Yaskawa INFORM job: X2_8B-21B(90,180).JBI

/JOB
//NAME X2_8B-21B(90,180)
///FOLDERNAME X2
//POS
///NPOS 939,939,939,42,0,0
///TOOL 0
///POSTYPE PULSE
///PULSE
C00000=1415,-134459,-133802,1969,12985,-79332
C00001=87080,-112473,-103627,41798,51237,-70410
C00002=91681,-107347,-99471,39221,49165,-68848
C00003=93439,-105106,-97054,38371,48113,-68361
C00004=93441,-104864,-95967,38672,47682,-68565
C00005=93504,-104969,-96260,38564,47753,-68495
C00006=95585,-102642,-95415,36914,47385,-67494
C00007=93504,-104969,-96260,38564,47753,-68495
C00008=87147,-112175,-102116,42180,50619,-70689
C00009=87145,-119394,-106475,25944,48524,-38750
C00010=91166,-110510,-101811,22693,48895,-36705
C00011=92650,-107060,-99920,21494,49065,-35962
C00012=94767,-104655,-99060,19829,49198,-34943
C00013=94484,-105085,-99259,20052,49173,-35080
C00014=93721,-102513,-96995,20598,49294,-35408
C00015=94484,-105085,-99259,20052,49173,-35080
C00016=89209,-117497,-105909,24366,48468,-37757
C00017=93166,-113214,-115710,1969,57926,-79332
C00018=93710,-106990,-108704,1652,56802,-79139
C00019=93766,-106412,-107148,1629,56140,-79127
C00020=93768,-106433,-106329,1638,55626,-79135
C00021=93918,-105383,-106173,1535,56065,-79069
C00022=94164,-101296,-104676,1361,57240,-78956
C00023=93895,-105502,-106499,1547,56205,-79076
C00024=93151,-113316,-114305,1998,57010,-79354
C00025=81072,-99391,-111155,4750,63110,-78553
C00026=81984,-95120,-104767,4287,61328,-78293
C00027=82103,-94682,-103397,4241,60705,-78273
C00028=82106,-94924,-102383,4271,59960,-78300
C00029=82089,-94934,-102578,4276,60076,-78302
C00030=82803,-90374,-100753,3806,61258,-77993
C00031=82089,-94934,-102578,4276,60076,-78302
C00032=81057,-100006,-109908,4804,62030,-78604
C00033=94004,-119945,-107122,-49530,42714,-48164
C00034=93972,-116281,-97047,-53343,39935,-45878
C00035=92833,-103149,-88492,-51302,40218,-47068
C00036=93174,-100930,-87132,-51219,40604,-47120
C00037=93174,-100493,-85792,-51770,40220,-46795
C00038=93174,-101015,-87399,-51095,40684,-47186
C00039=92955,-97894,-86230,-50180,41136,-47726
C00040=93303,-100448,-87190,-51023,40860,-47230
C00041=98055,-98607,-86499,-53149,43882,-46024
C00042=96642,-96320,-85623,-51883,43475,-46780
C00043=95342,-96864,-85830,-51299,42647,-47109
C00044=97130,-98187,-86063,-52744,43317,-46271
C00045=114545,-105110,-100746,-39625,57097,-48369
C00046=113947,-102413,-97570,-39574,56382,-48359
C00047=113947,-102278,-96691,-39772,56015,-48196
C00048=113346,-99976,-96570,-39024,56612,-48763
C00049=112899,-98120,-95866,-38597,56823,-49078
C00050=114020,-99555,-96940,-39169,57262,-48705
C00051=56302,-84822,-83054,58022,66572,-84014
C00052=58361,-85953,-83540,57558,65172,-83717
C00053=56302,-84822,-83054,58022,66572,-84014
C00054=50122,-85714,-86741,59061,71306,-84454
C00055=54195,-101901,-111197,24063,62262,-77343
C00056=67243,-111926,-101536,-21450,29925,-69540
C00057=66442,-101704,-94400,-19916,30532,-70304
C00058=66308,-99858,-92576,-19846,30336,-70336
C00059=66311,-99589,-91307,-20230,29731,-70137
C00060=66308,-99960,-93112,-19687,30597,-70418
C00061=70591,-100617,-92786,-25268,31264,-67678
C00062=70591,-100325,-91437,-25755,30647,-67424
C00063=68222,-99738,-91214,-22742,30105,-68906
C00064=70591,-100606,-92729,-25289,31242,-67667
C00065=66097,-110297,-96199,-21577,27345,-69446
C00066=65719,-107666,-92844,-21562,26575,-69447
C00067=65848,-106528,-92445,-21497,26927,-69482
C00068=65365,-110699,-93884,-21743,25627,-69354
C00069=67243,-111926,-101536,-21450,29925,-69540
C00070=68963,-41843,-96211,398,96948,48811
C00071=76932,-51697,-92360,-2602,89609,51106
C00072=71886,-45093,-85416,-705,88639,49643
C00073=71886,-45937,-84760,-705,87803,49648
C00074=71886,-44632,-85753,-705,89084,49641
C00075=68776,-90352,-95136,4313,51281,47645
C00076=68803,-86754,-93636,4241,52203,47695
C00077=68762,-92243,-95906,4353,50785,47617
C00078=77446,-64871,-91176,-8832,74282,49527
C00079=75907,-64612,-91046,-8095,74185,49034
C00080=78150,-64967,-91224,-9168,74335,49752
C00081=78150,-57569,-97635,-8943,81990,49191
C00082=68963,-41843,-96211,398,96948,48811
C00083=67385,-42511,-92598,992,94393,48367
C00084=66773,-44328,-90253,1220,92024,48175
C00085=66900,-44765,-89647,1171,91425,48205
C00086=66773,-43962,-90441,1221,92327,48178
C00087=69817,-49291,-93527,72,91467,49038
C00088=102407,-61387,-79216,-48101,75803,74984
C00089=99741,-62884,-79905,-47237,74215,74494
C00090=102407,-61387,-79216,-48101,75803,74984
C00091=71396,-101707,-96198,-105,39560,49678
C00092=71544,-99303,-95354,-247,40276,49753
C00093=71126,-105930,-97636,165,38275,49535
C00094=74447,-120283,-111838,-3099,39699,51260
C00095=57750,-84762,-113304,22338,79933,80646
C00096=38298,-117376,-123136,35520,84192,83183
C00097=31003,-114098,-105660,45955,85390,81321
C00098=32496,-116782,-107403,45795,84408,81579
C00099=34116,-118987,-108120,45640,83088,81742
C00100=33779,-118873,-108083,45678,83285,81673
C00101=33779,-118389,-106291,45736,82677,81394
C00102=33116,-116007,-107005,45711,84199,81779
C00103=35801,-87517,-89404,53765,81733,82681
C00104=39882,-82610,-88384,51436,81062,84322
C00105=41068,-84647,-89270,51225,80089,84396
C00106=40772,-84148,-89054,51277,80330,84378
C00107=40772,-84205,-87233,51414,79593,83963
C00108=38923,-82890,-88507,51652,81543,84094
C00109=36746,-57404,-73348,56767,88159,82454
C00110=45895,-41966,-67544,52307,91775,84594
C00111=46575,-44003,-68786,52133,91236,84629
C00112=46479,-43721,-68615,52158,91311,84624
C00113=46479,-44137,-67591,52124,90780,84319
C00114=45007,-43525,-68779,52515,92222,84403
C00115=28648,-44932,-73481,55068,103422,82059
C00116=23347,-70472,-95481,46672,94955,79134
C00117=23347,-70472,-95481,46672,94955,79134
C00118=34640,-80743,-102688,-17405,97112,73122
C00119=52690,-105642,-114364,-31889,95098,51390
C00120=51347,-103959,-112740,-31690,94497,51045
C00121=51347,-104280,-111882,-31650,93903,51212
C00122=54658,-102055,-112243,-32194,96275,51810
C00123=55140,-100848,-112208,-32308,96960,51798
C00124=56225,-98838,-109389,-32389,96760,52273
C00125=52710,-105778,-111943,-31798,93771,51772
C00126=54580,-102143,-110625,-32107,95358,52042
C00127=53574,-106836,-112314,-31893,93817,52092
C00128=52008,-102475,-110737,-31756,94333,51344
C00129=53574,-106836,-112314,-31893,93817,52092
C00130=61074,-96775,-114868,-33501,102293,52496
C00131=149084,-102156,-129577,-22032,95315,42360
C00132=128569,-114069,-129208,-14930,94899,36248
C00133=124702,-111484,-125119,-14131,93099,35189
C00134=123206,-111006,-122572,-13804,91571,34868
C00135=123205,-111346,-122108,-13798,91123,34918
C00136=123169,-110975,-122344,-13795,91444,34870
C00137=122647,-104244,-120003,-13724,93323,34489
C00138=123169,-110975,-122344,-13795,91444,34870
C00139=116503,-109521,-121739,-12400,90787,32743
C00140=113941,-110266,-121994,-11839,90202,31960
C00141=116503,-109521,-121739,-12400,90787,32743
C00142=121595,-114825,-128025,-13496,92670,34216
C00143=123984,-121300,-124584,-22039,85383,28695
C00144=118596,-113071,-118409,-20758,84424,26972
C00145=117828,-112575,-117002,-20585,83663,26833
C00146=117596,-112721,-116348,-20543,83158,26838
C00147=117643,-112201,-116474,-20543,83493,26797
C00148=117846,-106122,-114344,-20549,85245,26570
C00149=117643,-112201,-116474,-20543,83493,26797
C00150=125192,-113488,-115877,-22341,84450,29296
C00151=124919,-116220,-115928,-22323,83104,29449
C00152=122352,-116155,-116251,-21738,82647,28614
C00153=124919,-116220,-115928,-22323,83104,29449
C00154=123984,-121300,-124584,-22039,85383,28695
C00155=86442,-134681,-133724,19248,79211,32552
C00156=86002,-121949,-124889,19319,80358,32581
C00157=85994,-121959,-123892,19351,79775,32484
C00158=85995,-122137,-123177,19379,79272,32404
C00159=85938,-122450,-123568,19392,79360,32398
C00160=86651,-115539,-121342,19081,81262,32951
C00161=85938,-122450,-123568,19392,79360,32398
C00162=130270,-119263,-121891,-15868,79169,48216
C00163=132135,-133974,-122544,-16883,72658,49767
C00164=129371,-136174,-123179,-16117,71390,48932
C00165=132135,-133974,-122544,-16883,72658,49767
C00166=120611,-122953,-119681,-21560,80854,22535
C00167=120610,-122943,-118608,-21593,80243,22645
C00168=120610,-122853,-116921,-21650,79318,22813
C00169=120610,-122881,-117271,-21638,79506,22779
C00170=120610,-122878,-117279,-21638,79511,22778
C00171=120610,-122881,-117271,-21638,79506,22779
C00172=120610,-122873,-117198,-21640,79468,22785
C00173=120610,-122853,-117190,-21640,79473,22785
C00174=120610,-122873,-117198,-21640,79468,22785
C00175=120611,-122910,-120952,-21522,81605,22399
C00176=120612,-120891,-127143,-3106,87300,4415
C00177=120611,-122177,-124352,-3111,84925,4474
C00178=120611,-122645,-122467,-3116,83527,4507
C00179=120611,-122779,-121606,-3119,82929,4523
C00180=120611,-122697,-122159,-3117,83311,4513
C00181=120611,-122692,-122166,-3117,83318,4513
C00182=120611,-122697,-122159,-3117,83311,4513
C00183=120611,-121412,-126223,-3107,86468,4436
C00184=96873,-136971,-131305,-19961,95014,27830
C00185=53188,-122774,-119059,-34227,101931,42117
C00186=53187,-122644,-116623,-34032,100735,42492
C00187=53184,-122447,-115007,-33919,99986,42724
C00188=53180,-122268,-113886,-33849,99484,42877
C00189=53186,-122531,-115629,-33961,100272,42636
C00190=53233,-122033,-113114,-32057,113501,44659
C00191=53229,-122037,-113108,-32057,113495,44659
C00192=53233,-122033,-113114,-32057,113501,44659
C00193=53127,-122157,-112856,-34567,84618,41563
C00194=53132,-122146,-112848,-34568,84621,41564
C00195=53127,-122157,-112856,-34567,84618,41563
C00196=53124,-122720,-116247,-34514,86111,41098
C00197=68676,-133744,-131015,-10578,108811,68614
C00198=80160,-118182,-130261,41,125141,81817
C00199=80187,-122370,-123619,70,118933,81856
C00200=80183,-122639,-122398,68,118043,81854
C00201=80181,-122756,-121636,67,117515,81853
C00202=80184,-122603,-122588,68,118179,81854
C00203=80182,-122615,-122584,67,118170,81853
C00204=80184,-122603,-122588,68,118179,81854
C00205=80200,-121154,-126606,75,121396,81862
C00206=109164,-117358,-132635,7350,119146,48306
C00207=144183,-119511,-130571,15498,107286,7245
C00208=197934,-122815,-127402,28006,89082,-55776
C00209=202772,-123889,-124791,27048,85608,-54814
C00210=204705,-124106,-122314,26692,83530,-54575
C00211=204705,-124189,-120905,26732,82711,-54762
C00212=205113,-122699,-120601,26621,83104,-54520
C00213=208506,-122040,-120392,25870,82241,-53457
C00214=204510,-125657,-121990,26775,82699,-54838
C00215=204510,-125393,-124777,26704,84359,-54459
C00216=217123,-144581,-130617,26990,80795,-43719
C00217=208514,-157553,-136215,22784,79668,-13108
C00218=208514,-151468,-127497,22936,77598,-13510
C00219=209226,-147410,-126429,22728,78719,-13024
C00220=208514,-151468,-127497,22936,77598,-13510
C00221=208514,-156517,-134755,22805,79329,-13174
C00222=187736,-116553,-120968,36188,98329,-31010
C00223=144869,-104708,-130913,-697,92502,12445
C00224=97478,-100538,-119508,-25976,122096,72949
C00225=94415,-115583,-120723,-24602,114867,73486
C00226=94145,-116737,-119872,-24403,113768,73630
C00227=94090,-116915,-118863,-24267,113100,73760
C00228=94227,-118887,-121662,-24392,113788,73658
C00229=94618,-126072,-123928,-23885,111795,74261
C00230=93811,-121058,-122280,-24303,112998,73673
C00231=123165,-134656,-120887,-30393,109989,65140
C00232=122877,-135920,-118822,-30065,108215,65520
C00233=120918,-135771,-118381,-30417,107339,64954
C00234=122877,-135920,-118822,-30065,108215,65520
C00235=123434,-129548,-123417,-31323,113703,64157
C00236=126606,-101457,-128935,-16844,101795,36174
C00237=152779,-135138,-131563,-2515,76140,19155
C00238=150820,-122490,-124749,-1875,78392,18455
C00239=150097,-118368,-121531,-1645,78513,18212
C00240=150095,-118599,-120646,-1648,77850,18220
C00241=147666,-112236,-119185,-871,80184,17389
C00242=146670,-110099,-118456,-556,80825,17059
C00243=148658,-114325,-119887,-1186,79554,17722
C00244=87079,-91764,-103818,42328,107533,-9448
C00245=87027,-91004,-101788,42122,106912,-9740
C00246=89264,-90509,-101588,42089,105978,-9119
C00247=87027,-91004,-101788,42122,106912,-9740
C00248=87391,-90282,-107909,43186,109836,-8282
C00249=92115,-87061,-118989,19004,94950,3823
C00250=78975,-130870,-123203,-19746,71053,12291
C00251=74317,-97013,-111518,-17407,83606,9286
C00252=74211,-95430,-110119,-17377,83539,9259
C00253=74211,-95892,-109317,-17397,82840,9358
C00254=75305,-113551,-114600,-17838,69768,10493
C00255=78326,-111051,-111958,-19079,70114,11550
C00256=78379,-106110,-110225,-18937,71523,11339
C00257=78263,-116865,-113913,-19272,68408,11810
C00258=85880,-113569,-112821,-22054,71256,14152
C00259=85920,-114580,-110580,-22309,69503,14507
C00260=82054,-114988,-110714,-20879,68380,13249
C00261=85920,-114580,-110580,-22309,69503,14507
C00262=78975,-130870,-123203,-19746,67177,12291
C00263=159950,-115131,-126913,23322,109234,-64770
C00264=163413,-124246,-126581,22686,103792,-64589
C00265=164859,-127477,-125491,22457,101245,-64551
C00266=164857,-127553,-124648,22406,100728,-64651
C00267=164862,-127370,-126252,22506,101730,-64457
C00268=158275,-145382,-129341,21795,96649,-67831
C00269=159759,-153222,-131425,21726,93697,-67826
C00270=158275,-145382,-129341,21795,96649,-67831
C00271=157577,-144643,-126617,21696,95625,-68274
C00272=160219,-140867,-125578,21868,96138,-67212
C00273=157577,-144643,-126617,21696,95625,-68274
C00274=152631,-134238,-128202,21932,102817,-68768
C00275=146941,-123801,-133763,3444,102850,-52685
C00276=136178,-116173,-124987,-31736,84906,-22811
C00277=134413,-106132,-117362,-31242,84680,-23412
C00278=134231,-105594,-115694,-31219,83968,-23286
C00279=134230,-105863,-115134,-31239,83552,-23172
C00280=134007,-104199,-114803,-31151,84035,-23389
C00281=133473,-100630,-113499,-30965,84737,-23780
C00282=134315,-106237,-115533,-31260,83629,-23161
C00283=136272,-117460,-124003,-31807,83855,-22481
C00284=136226,-116324,-125056,-31750,84893,-22789
C00285=134474,-106353,-117504,-31259,84679,-23389
C00286=134275,-105758,-115681,-31235,83904,-23252
C00287=134274,-105987,-115198,-31252,83547,-23154
C00288=134027,-104733,-115029,-31162,83924,-23350
C00289=133465,-100971,-113658,-30966,84667,-23763
C00290=134308,-106598,-115693,-31262,83551,-23142
C00291=136269,-117902,-124178,-31812,83752,-22453
C00292=139753,-124875,-130430,-383,75663,26245
C00293=143223,-157944,-133481,5653,58679,38405
C00294=140983,-144085,-126452,6488,61628,37698
C00295=140148,-138933,-122655,6835,62006,37402
C00296=140147,-138616,-121921,6853,61719,37384
C00297=140691,-136506,-121897,6553,62737,37651
C00298=138669,-131542,-120459,7325,64564,37004
C00299=140691,-136506,-121897,6553,62737,37651
C00300=145148,-139028,-124584,4588,62787,39337
C00301=159973,-92454,-110285,-14523,90938,48717
C00302=158765,-97223,-112137,-14224,89465,48492
C00303=159973,-92454,-110285,-14523,90938,48717
C00304=164681,-91509,-114703,-15696,94847,49769
C00305=142525,-105883,-132766,7713,103357,60336
C00306=90751,-115691,-121566,36045,104861,61043
C00307=92920,-122587,-117773,35137,99152,60047
C00308=93124,-123070,-117553,35091,98753,60003
C00309=93124,-123008,-116878,35050,98435,59900
C00310=93160,-123063,-117190,35068,98555,59953
C00311=95752,-125144,-117838,34977,96947,60505
C00312=93160,-123063,-117190,35068,98555,59953
C00313=92038,-109836,-114685,38536,89453,57060
C00314=86810,-100893,-104585,47463,92019,56975
C00315=88449,-102594,-103600,47188,90148,56855
C00316=88449,-102618,-102426,47172,89639,56610
C00317=88449,-102603,-103366,47184,90046,56806
C00318=85133,-99388,-102162,47637,92393,56350
C00319=85168,-99488,-101153,47595,91912,56132
C00320=86978,-101259,-101820,47360,90627,56378
C00321=84037,-98201,-102123,47804,93363,56297
C00322=108771,-112096,-123986,16313,85813,59347
C00323=109769,-112695,-132242,3132,99947,61138
C00324=127404,-127157,-120795,-27540,73197,60883
C00325=120526,-123085,-115007,-25540,69700,59025
C00326=119461,-122312,-114032,-25210,69192,58723
C00327=119461,-122116,-113003,-25293,68708,58832
C00328=119461,-122312,-114032,-25210,69192,58723
C00329=94655,-112249,-115827,1041,75214,51009
C00330=93364,-111129,-115444,1499,75574,50577
C00331=121213,-123445,-114215,-25873,69302,59387
C00332=127714,-127278,-119628,-27738,72603,61150
C00333=140848,-129628,-128054,-17424,84805,27418
C00334=127903,-106251,-120637,-17388,91568,15860
C00335=124887,-98361,-114445,-16717,91208,14907
C00336=124614,-94849,-112077,-16660,91489,14780
C00337=117832,-103976,-115449,-15062,87719,13014
C00338=118209,-109888,-118953,-15141,86934,13233
C00339=120968,-118649,-124805,-15800,86569,14208
C00340=112726,-101228,-128594,-1890,90279,-15897
C00341=102865,-105549,-130121,1361,88970,-18873
C00342=85416,-143080,-122146,23399,58401,-32529
C00343=89847,-131888,-116792,20882,59491,-30436
C00344=92362,-125061,-113696,19444,60385,-29236
C00345=93061,-123120,-113350,17672,61903,-28193
C00346=94553,-118505,-112300,14045,65420,-26024
C00347=98668,-108930,-110937,8182,72602,-22159
C00348=97558,-114678,-114533,8498,72116,-22521
C00349=94805,-124749,-120489,9597,70928,-23580
C00350=89899,-115674,-129227,15589,81503,-27304
C00351=94000,-113154,-130859,-1035,116659,75004
C00352=93721,-118000,-129934,-5060,122177,74127
C00353=93715,-120352,-127357,-4900,119392,74256
C00354=95323,-119775,-124837,-4467,118233,74917
C00355=88228,-120746,-125279,-6046,117555,72254
C00356=93725,-120284,-127319,-4898,119404,74259
C00357=93731,-117931,-129895,-5059,122189,74130
C00358=92605,-107385,-114202,42080,118626,78084
C00359=94957,-117308,-114744,40643,113912,77125
C00360=98035,-118959,-113942,40650,111458,77555
C00361=97377,-118969,-113658,40508,111623,77311
C00362=92838,-119913,-111612,39284,112339,75456
C00363=89330,-129662,-113469,38848,107684,75257
C00364=90618,-118755,-112828,39302,114392,75239
C00365=88476,-109244,-112462,40625,118981,76164
C00366=73726,-95231,-122050,23824,117115,78775
C00367=68964,-113071,-130294,-19412,109419,80322
C00368=55630,-112625,-122011,-35520,97927,81697
C00369=52390,-118820,-120628,-34805,93310,81881
C00370=47903,-104132,-115503,-31781,99116,78849
C00371=50154,-103283,-114443,-33074,100204,79243
C00372=58838,-110339,-112590,-36869,98506,82639
C00373=58731,-119232,-119174,-35403,94943,83913
C00374=59872,-116629,-120975,-35716,97415,83571
C00375=61517,-148095,-119735,-48293,75564,80066
C00376=56687,-146008,-116451,-48020,72337,79248
C00377=54787,-145656,-114853,-48003,70776,79074
C00378=55742,-144545,-112808,-48270,70818,79550
C00379=55476,-147094,-115701,-48129,70996,79318
C00380=61520,-147186,-118480,-48348,75358,80173
C00381=69196,-132761,-125763,-48066,87564,77891
C00382=67178,-112107,-133350,9560,121946,71499
C00383=53652,-115588,-130730,10921,119132,80041
C00384=53631,-118653,-128170,10572,116038,79726
C00385=49979,-127897,-130457,9357,109364,77840
C00386=56749,-116857,-125794,10963,115112,80794
C00387=55258,-116620,-125691,10759,115364,80266
C00388=57875,-118021,-126871,3069,115075,80163
C00389=60441,-120565,-127584,-682,114000,80575
C00390=56047,-119336,-124870,-1283,112953,79038
C00391=53493,-120154,-126714,-1639,113579,78070
C00392=53512,-117734,-129516,-1682,116546,78033
C00393=64263,-112177,-127274,-18013,116425,52133
C00394=53349,-113292,-116223,-34708,105130,41711
C00395=53347,-113647,-113946,-34435,103813,42137
C00396=52619,-113100,-112715,-34376,103127,42055
C00397=57761,-122997,-112011,-36249,97635,45734
C00398=53343,-113729,-112902,-34324,103242,42318
C00399=53345,-113489,-115217,-34581,104530,41905
C00400=83368,-135406,-127982,-43757,111124,-24122
C00401=107112,-148704,-121184,-48737,110155,-73723
C00402=107085,-142005,-111593,-48000,108472,-72828
C00403=107084,-140010,-108705,-47787,107957,-72557
C00404=87341,-136498,-115496,-38254,104619,-81025
C00405=107242,-151301,-127119,1131,113743,-57617
C00406=97067,-157300,-128671,2718,111508,-55981
C00407=110320,-141463,-116471,39094,91497,-45920
C00408=107133,-145289,-116877,40503,90261,-47122
C00409=107139,-146938,-119316,40521,90762,-46927
C00410=81304,-146505,-131302,46256,99624,-33732
C00411=42290,-135810,-134986,6789,56953,43412
C00412=53482,-111499,-99357,5283,31563,44884
C00413=53488,-110753,-96932,5448,30458,44798
C00414=53767,-110832,-96596,5125,30193,44961
C00415=53784,-109802,-93724,5302,28956,44868
C00416=54077,-108600,-90505,5126,27581,44957
C00417=54077,-108600,-90505,5126,27581,44957
C00418=53472,-108968,-91791,5862,28222,44586
C00419=53466,-109889,-94290,5675,29282,44681
C00420=93748,-113667,-111432,-27227,62688,41579
C00421=93751,-113561,-109328,-27520,61581,41869
C00422=94298,-111463,-107612,-27765,61782,42046
C00423=94581,-111188,-102370,-28702,59144,42896
C00424=93743,-112935,-104615,-28181,59286,42489
C00425=93741,-113330,-106821,-27872,60309,42206
C00426=53707,-103235,-126817,3349,90409,72793
C00427=53694,-107630,-124107,3352,86490,72685
C00428=54249,-109117,-122940,3188,84989,72821
C00429=53889,-108493,-122718,3296,85190,72712
C00430=53934,-108401,-122669,3281,85203,72729
C00431=53898,-108487,-122690,3292,85171,72715
C00432=53735,-107561,-124050,3339,86489,72698
C00433=53748,-103173,-126762,3336,90406,72805
C00434=24309,-104032,-127063,11845,92683,63842
C00435=14692,-96968,-103634,28347,84848,56264
C00436=69737,67118,16632,42575,112328,80617
C00437=69765,65699,24866,49286,110081,81190
C00438=67763,57248,15205,49930,112177,81338
C00439=66597,45471,2237,49732,108456,84264
C00440=65732,29116,-14706,47956,102511,88210
C00441=64654,15507,-27591,48359,103674,88304
C00442=64160,11579,-31342,48521,104111,88301
C00443=61960,-11325,-50587,48960,105231,87855
C00444=62752,-490,-42039,50927,111117,85502
C00445=59065,9442,-33802,52095,101706,84381
C00446=72891,31150,-30442,36756,97726,81673
C00447=90877,-16324,-74885,22437,92008,81813
C00448=102330,-22799,-82036,-11222,88832,73278
C00449=48313,-118911,-129560,-19207,92704,27073
C00450=53495,-110604,-121584,-20154,93282,28749
C00451=52758,-114738,-121214,-19966,90894,28894
C00452=53577,-108529,-119024,-20154,92819,28853
C00453=53441,-111570,-120070,-20107,91929,28955
C00454=54259,-112639,-122766,-20278,93161,29031
C00455=53522,-108468,-123882,-20258,95652,28360
C00456=66910,-101677,-117691,-1645,82254,-17515
C00457=66905,-103395,-115374,-1652,79946,-17486
C00458=66781,-102668,-113970,-1597,79454,-17514
C00459=66805,-103111,-114336,-1620,79451,-17514
C00460=68500,-103754,-114391,-2206,79196,-16952
C00461=69944,-105966,-109421,-11944,70678,-17306
C00462=66783,-105788,-110032,-11324,70201,-18483
C00463=66785,-105108,-112553,-11207,72068,-18659
C00464=34610,-119076,-126707,31995,89279,-47352
C00465=26693,-119602,-105841,51320,82883,-62074
C00466=26676,-118953,-103885,51392,82336,-62389
C00467=27513,-117883,-103390,51295,82023,-62119
C00468=27155,-116250,-99936,51446,81403,-62657
C00469=26666,-118021,-101324,51491,81640,-62785
C00470=26683,-118745,-103309,51412,82173,-62476
C00471=26741,-121947,-116429,51038,86269,-60171
C00472=80158,-111738,-121779,46707,81282,33331
C00473=80124,-114295,-114082,47454,77096,31277
C00474=80115,-114367,-110881,47781,75720,30584
C00475=82694,-112805,-110607,45433,76546,32096
C00476=79416,-116776,-110373,48221,75031,29878
C00477=80052,-114603,-110983,47806,75713,30548
C00478=80061,-114542,-114188,47480,77086,31241
C00479=80063,-113108,-120040,30435,104055,77976
C00480=80050,-114212,-116860,30086,101864,77373
C00481=79953,-112412,-114936,30056,101673,77283
C00482=79896,-114545,-111990,35011,85373,77209
C00483=80002,-114499,-112021,34994,85367,77250
C00484=80418,-112503,-109508,36583,80313,77299
C00485=80029,-114714,-111597,36713,80437,77233
C00486=82440,-93132,-104306,35744,84828,79668
C00487=83142,-90791,-100833,35602,83775,79606
C00488=86899,-75258,-94009,34443,85431,81601
C00489=81341,-82881,-101909,35963,88366,80388
C00490=80042,-114535,-115070,36542,82240,77847
C00491=80040,-111621,-122742,8414,85267,41918
C00492=80035,-113457,-119567,8450,82400,41723
C00493=81653,-127299,-120603,7413,72175,41563
C00494=80787,-111090,-118654,-2680,86591,53574
C00495=79816,-113282,-119312,-2452,85841,53272
C00496=79371,-114754,-119577,-3684,84607,55046
C00497=80002,-113603,-119620,-10752,83390,63441
C00498=80006,-103113,-128729,-10775,94202,62513
C00499=39776,-103787,-110683,21075,62663,-59255
C00500=39766,-104399,-107995,21452,60825,-59622
C00501=42409,-98411,-106612,17292,64181,-58311
C00502=40224,-103973,-106702,21316,60174,-59568
C00503=40236,-103975,-106617,21326,60117,-59576
C00504=39744,-104425,-108009,21464,60826,-59630
C00505=39754,-103814,-110697,21087,62664,-59263
C00506=47977,-106691,-119962,23629,83327,-62671
C00507=66867,-99660,-121232,22132,99220,-62132
C00508=66851,-102572,-118810,21937,96446,-62653
C00509=75734,-133384,-127933,14237,79030,-52956
C00510=72894,-135572,-127272,15029,78051,-54067
C00511=68354,-138260,-126704,16229,77252,-55778
C00512=51043,-132166,-118737,30188,81179,-60892
C00513=66851,-103895,-117201,21852,94891,-62938
C00514=66868,-101493,-119792,22004,97521,-62449
C00515=74321,-107832,-126985,-11736,80239,-61811
C00516=66584,-114412,-108983,-34198,49386,-64476
C00517=66581,-113854,-105403,-35147,47795,-63826
C00518=60037,-123864,-103215,-32979,33373,-60846
C00519=66685,-112635,-100589,-36483,45924,-62949
C00520=66087,-122535,-98001,-45910,35159,-56780
C00521=66087,-122589,-97589,-46197,34963,-56624
C00522=66567,-113311,-102857,-35821,46729,-63375
C00523=66569,-114089,-106515,-34851,48256,-64025
C00524=66614,-114312,-115902,-32344,53032,-65825
C00525=26293,-124733,-123676,-35115,86081,-77095
C00526=26278,-124914,-120130,-35186,84196,-76502
C00527=26896,-123210,-118103,-35309,84144,-76233
C00528=26306,-121290,-117658,-35177,84490,-76583
C00529=26301,-124893,-120124,-35190,84211,-76498
C00530=26317,-124710,-123669,-35119,86096,-77090
C00531=26368,-124828,-121889,-39154,95960,-78120
C00532=26350,-124746,-118556,-38992,94373,-77544
C00533=26743,-123924,-117047,-38976,94149,-77295
C00534=25994,-118731,-112182,-38918,93559,-77400
C00535=26347,-124286,-115407,-38884,93032,-77056
C00536=26365,-124761,-118865,-39006,94524,-77592
C00537=26264,-124528,-116402,-47920,86072,-68134
C00538=26249,-123768,-112787,-47988,84810,-67516
C00539=26243,-123374,-111311,-48022,84325,-67278
C00540=27566,-121809,-108978,-48187,84599,-66758
C00541=26232,-123227,-110778,-48035,84146,-67194
C00542=26247,-124165,-114452,-47952,85370,-67795
C00543=82585,-123093,-118421,-52491,64599,-59558
C00544=107155,-118824,-102398,-58122,50036,-52281
C00545=107155,-117467,-98958,-59145,49269,-51564
C00546=97405,-116506,-103900,-42249,48003,-50997
C00547=106070,-119659,-109558,-10435,43390,-62985
C00548=106582,-120227,-109824,-10893,43331,-62728
C00549=108221,-120478,-109947,-12283,43512,-61940
C00550=107366,-119665,-105766,-8068,39033,-71395
C00551=107169,-120346,-107141,-7797,39493,-71540
C00552=108433,-119625,-117514,-7930,46308,-71537
C00553=107111,-122100,-111275,-39348,45202,-56077
C00554=107109,-117760,-98763,-43179,41028,-53713
C00555=107588,-117193,-97805,-43718,41045,-53392
C00556=106524,-118597,-102582,-12234,37369,-61918
C00557=94589,-117778,-102277,12815,37699,-75547
C00558=102638,-119985,-97555,45693,41122,-79392
C00559=107127,-114270,-91297,56630,43098,-80056
C00560=101354,-119078,-102486,55464,49091,-79315
C00561=93612,-109275,-133010,-12113,75674,-64968
C00562=74458,-81913,-116300,-25886,107898,-47202
C00563=74285,-84923,-113224,-25351,104735,-46539
C00564=81136,-80920,-107787,-32217,106507,-45804
C00565=73205,-70766,-105026,-26930,108371,-55320
C00566=67013,-54988,-96314,-28913,109390,-56440
C00567=64326,-60619,-98517,-27945,103439,-54917
C00568=60588,-58283,-100875,-23679,106756,-51616
C00569=60637,-54628,-103477,-24231,109960,-52288
C00570=76657,-70403,-83915,-51355,64349,-40407
C00571=74830,-68241,-74355,-53953,55282,-38932
C00572=73110,-62379,-68708,-53436,54020,-39148
C00573=73205,-61459,-68120,-53411,54142,-39173
C00574=37101,-67408,-75626,25719,44355,-77225
C00575=80454,-89253,-85222,-18196,36589,-55164
C00576=82537,-90732,-84998,-19061,34673,-56543
C00577=81508,-95500,-88175,-18158,33969,-56993
C00578=81043,-103588,-94156,-17854,33413,-57140
C00579=82846,-88179,-88219,-41798,48730,-43563
C00580=81818,-81213,-82326,-41198,48211,-43888
C00581=79628,-80184,-80995,-37948,46295,-45131
C00582=64054,-84747,-85294,-4301,39779,-58682
C00583=75679,-87820,-86686,-15780,40506,-52732
C00584=49490,-70910,-80897,34287,57978,-66074
C00585=46339,-68382,-80235,37741,61555,-66618
C00586=42699,-70655,-83815,39176,63943,-67342
C00587=43803,-67144,-92021,36183,69839,-64523
C00588=86906,-70734,-117845,-25978,101850,-24881
C00589=194376,-118372,-116958,-36622,58194,75254
C00590=187943,-106127,-101715,-33777,52366,74665
C00591=187951,-105693,-98645,-34509,50978,75202
C00592=188084,-106418,-97655,-35041,50218,75578
C00593=188317,-106012,-97596,-35084,50459,75600
C00594=188444,-106426,-98768,-20061,46138,60546
C00595=187923,-105820,-99644,-19403,46817,60144
C00596=187914,-106157,-102495,-18928,48312,59826
C00597=188021,-109107,-91072,-54887,40419,77132
C00598=188025,-108188,-88773,-55807,39869,77674
C00599=188027,-107805,-87846,-56180,39654,77892
C00600=188036,-107761,-87717,-56242,39627,77928
C00601=188035,-108145,-88644,-55869,39841,77710
C00602=188030,-109068,-90945,-54948,40390,77168
C00603=188015,-114130,-110744,-41340,72657,75143
C00604=188018,-113864,-107763,-41683,71368,75679
C00605=188019,-113684,-106544,-41824,70871,75888
C00606=188009,-113674,-106577,-41816,70886,75877
C00607=188008,-113852,-107795,-41674,71383,75668
C00608=188005,-114114,-110775,-41332,72673,75132
C00609=187933,-113872,-110928,-18210,58720,57176
C00610=187882,-113256,-105308,719,43762,42538
C00611=187896,-112711,-102669,725,42418,42533
C00612=188420,-113689,-102063,268,41535,42791
C00613=188115,-112866,-98519,1306,37390,42477
C00614=187899,-111729,-99017,1491,38283,42378
C00615=187886,-112431,-101600,1465,39511,42393
C00616=192869,-127835,-120494,-22551,66263,53872
C00617=188079,-122619,-114609,-40714,83609,61664
C00618=188077,-122103,-112045,-40794,82601,62056
C00619=187715,-122511,-111198,-41935,87054,59703
C00620=187919,-121855,-110458,-41952,87063,59791
C00621=187909,-121652,-109146,-41964,86526,60005
C00622=188106,-121566,-109755,-41972,86936,59927
C00623=188110,-122188,-112187,-41960,87826,59570
C00624=188058,-121965,-125191,-40549,88870,59628
C00625=104402,-90439,-123637,-22599,88102,-26907
C00626=80407,-121901,-119741,-18448,66455,-46046
C00627=80400,-121844,-116068,-18757,64334,-45697
C00628=80537,-121388,-114459,-18932,63649,-45528
C00629=79603,-120238,-114067,-18464,63768,-45911
C00630=80475,-121542,-115946,-18779,64427,-45684
C00631=80482,-121578,-119613,-18469,66554,-46034
C00632=85156,-144709,-129107,21632,59402,-64028
C00633=93856,-120445,-109825,39450,57641,-70752
C00634=92040,-118150,-105716,42198,57852,-71483
C00635=84290,-104454,-97866,49611,66426,-72991
C00636=89339,-123311,-104077,50362,59795,-74015
C00637=89538,-124434,-104337,50489,59412,-74133
C00638=89538,-124434,-104337,50489,59412,-74133
C00639=93820,-118277,-102341,40471,46353,-72255
C00640=93828,-119232,-105178,39715,47322,-71755
C00641=93822,-120125,-107980,28359,52237,-38282
C00642=93816,-119582,-106091,28689,51458,-38525
C00643=93586,-119120,-105470,28875,51409,-38650
C00644=93805,-118409,-102529,29499,49391,-39302
C00645=93820,-119862,-107056,29266,59584,-40856
C00646=93823,-120114,-107958,29147,59957,-40747
C00647=93830,-120670,-110185,28854,60909,-40473
C00648=63807,-119595,-131717,32346,77391,-31957
C00649=66677,-122882,-119460,9954,65715,31882
C00650=66675,-122709,-116301,10101,63887,31721
C00651=67233,-123478,-115304,9930,62823,31836
C00652=66931,-123352,-121183,-9496,81515,37764
C00653=66923,-123307,-121544,-9492,81753,37743
C00654=68643,-124975,-117174,-29306,103015,42901
C00655=66675,-122499,-114776,-33395,107690,42822
C00656=66677,-122795,-117228,-33681,108831,42458
C00657=66720,-122114,-124411,-34847,112827,41144
C00658=15972,-110889,-128286,10965,59905,43045
C00659=15972,-110889,-128286,10965,59905,43045
C00660=101389,-60822,-75148,-6919,68546,70102
C00661=115790,69230,64798,8053,66131,71909
C00662=120688,105020,73307,12402,84846,73777
C00663=120868,103639,75593,12409,82749,73629
C00664=115729,87511,60668,24910,80664,72140
C00665=115729,87728,62416,24969,79785,71953
C00666=115729,87559,61087,24923,80450,72095
C00667=115791,92601,67435,24996,79233,71857
C00668=115791,92884,68992,25055,78493,71699
C00669=115775,91432,67152,25030,78849,71769
C00670=115791,92590,67368,24993,79266,71865
C00671=126095,92435,63058,5152,80409,74477
C00672=126453,92655,64525,5082,79598,74565
C00673=125768,92396,64197,5232,79709,74335
C00674=126453,92544,63242,5072,80328,74595
C00675=120228,112105,88453,12614,79365,73063
C00676=120053,112844,85327,12571,81642,73235
C00677=120830,71540,61874,4756,55589,66514
C00678=120535,76858,72419,5134,51864,66212
C00679=120418,79487,77321,5314,50212,66075
C00680=120418,81305,81326,5435,48689,65991
C00681=120418,79487,77321,5314,50212,66075
C00682=121101,73566,71896,4942,50464,66384
C00683=120640,77942,77238,5256,49458,66131
C00684=121101,73566,71896,4942,50464,66384
C00685=121222,71175,67349,4775,52021,66512
C00686=121527,63287,45853,4167,61152,67017
C00687=121222,53388,35819,-506,60999,72680
C00688=120886,47658,32975,-2750,58873,75677
C00689=120357,43570,36815,-5865,53609,79607
C00690=120357,44263,39245,-5952,52477,79673
C00691=120357,43570,36815,-5865,53609,79607
C00692=121171,39511,33217,-6288,53799,79936
C00693=121171,39929,34748,-6347,53075,79981
C00694=120657,42834,37803,-6102,52651,79790
C00695=121171,39929,34748,-6347,53075,79981
C00696=121307,38577,31710,-6326,54255,79965
C00697=121648,35573,24568,-6294,57116,79932
C00698=109578,65571,33028,8923,84264,70984
C00699=101389,-60822,-75148,-6919,68546,70102
C00700=96929,-90691,-89138,-5080,61517,23019
C00701=109818,-91701,-74936,-12505,53754,-21374
C00702=124678,-6429,-38037,-6148,92089,-49038
C00703=133997,38575,-5386,-4879,105902,-64390
C00704=134430,35731,-4221,-4855,103756,-64161
C00705=134605,34666,-3678,-4847,102887,-64068
C00706=134604,34193,-2477,-4825,101908,-64030
C00707=134605,34666,-3678,-4847,102887,-64068
C00708=133324,38381,1851,-4717,101326,-64430
C00709=133984,36157,-436,-4773,101627,-64224
C00710=133324,38381,1851,-4717,101326,-64430
C00711=132740,42105,45,-4739,104308,-64739
C00712=149381,11612,-10676,-29411,77480,-58612
C00713=147438,22168,3080,-29176,74144,-58502
C00714=146667,27061,10007,-29185,72341,-58335
C00715=146666,27163,11157,-29282,71765,-58183
C00716=146667,27014,9351,-29131,72675,-58422
C00717=147917,24004,8167,-29618,72393,-57848
C00718=149025,12105,-2903,-29837,73391,-57674
C00719=148491,19843,4212,-29741,72852,-57742
C00720=149112,19141,-2052,-29482,76126,-58364
C00721=148788,18564,-14441,-28797,82460,-60100
C00722=147017,27605,-1759,-28452,79091,-59917
C00723=146805,27803,661,-28506,77793,-59674
C00724=146803,27699,1600,-28565,77235,-59535
C00725=146805,27874,109,-28472,78126,-59757
C00726=148390,24338,-1607,-29025,77984,-59121
C00727=147556,26192,183,-28786,77573,-59333
C00728=148390,24338,-1607,-29025,77984,-59121
C00729=149162,23542,-7999,-28991,81344,-59682
C00730=129846,-17397,-52274,-16165,101048,-68229
C00731=103949,-6271,-30701,-7884,96105,-76175
C00732=94102,16895,-5866,-4380,94047,-79161
C00733=94024,14878,-3719,-4358,91692,-79105
C00734=93993,14152,-2780,-4351,90742,-79083
C00735=93993,14253,-1030,-4349,89719,-79047
C00736=93993,14152,-2780,-4351,90742,-79083
C00737=93685,20015,4382,-4321,89334,-79138
C00738=93881,17120,1686,-4338,89515,-79078
C00739=93685,20015,4382,-4321,89334,-79138
C00740=93796,22544,1176,-4343,92603,-79213
C00741=95224,-25687,-42365,-27028,60157,-72238
C00742=94111,-23276,-36997,-26973,57954,-72128
C00743=93676,-22245,-34794,-26967,57075,-72081
C00744=93677,-22196,-33100,-27266,56165,-71832
C00745=93676,-22245,-34794,-26967,57075,-72081
C00746=94165,-26445,-35973,-27662,55954,-71554
C00747=93910,-23559,-33944,-27450,56079,-71704
C00748=94165,-26445,-35973,-27662,55954,-71554
C00749=95768,-30118,-43626,-27714,58991,-71694
C00750=97625,-41604,-59467,-17173,89706,8843
C00751=96114,-37688,-53918,-16886,88057,8555
C00752=95526,-36022,-51615,-16777,87400,8443
C00753=95527,-36150,-50037,-16784,86406,8579
C00754=95526,-36022,-51615,-16777,87400,8443
C00755=95532,-36183,-50637,-16782,86745,8534
C00756=95234,-33170,-48668,-16723,87008,8396
C00757=95532,-36183,-50637,-16782,86745,8534
C00758=95504,-36095,-50208,-16778,86530,8554
C00759=93996,-36675,-50581,-16493,86163,8084
C00760=95504,-36095,-50208,-16778,86530,8554
C00761=97625,-41604,-59467,-17173,89706,8843
C00762=101873,-77751,-87156,-42969,63075,-62474
C00763=95937,-74809,-81328,-40948,58735,-63434
C00764=95565,-74583,-80935,-40815,58468,-63500
C00765=95566,-74620,-79294,-41227,57681,-63141
C00766=95565,-74583,-80935,-40815,58468,-63500
C00767=98755,-73227,-80296,-42221,60183,-62682
C00768=98803,-73638,-78797,-42678,59356,-62269
C00769=96868,-74481,-79195,-41849,58298,-62761
C00770=98803,-73638,-78797,-42678,59356,-62269
C00771=97163,-69666,-76891,-41573,59236,-63045
C00772=96752,-66139,-75134,-41097,59602,-63417
C00773=97163,-69666,-76891,-41573,59236,-63045
C00774=101873,-77751,-87156,-42969,63075,-62474
C00775=126113,-49786,-51573,-51544,90004,-55144
C00776=123973,-50127,-48217,-51392,87374,-54806
C00777=123267,-50126,-46982,-51347,86566,-54726
C00778=118449,-34614,-37258,-50921,85079,-56444
C00779=119272,-35479,-39244,-50973,86038,-56539
C00780=121232,-35158,-42579,-51146,88553,-56901
C00781=111145,-57425,-62081,-41633,61582,-55088
C00782=109620,-53993,-56645,-41578,59663,-54986
C00783=109182,-52175,-54253,-41602,59047,-54926
C00784=105694,-54761,-55728,-40263,57099,-55829
C00785=106107,-56401,-57979,-40230,57706,-55889
C00786=107578,-60042,-63488,-40293,59558,-55964
C00787=93331,-25535,-46307,-22677,87971,-72102
C00788=84242,-5399,-27465,-11713,100257,-81196
C00789=83743,-8192,-25851,-11599,97806,-81134
C00790=83568,-8790,-24556,-11558,96698,-81088
C00791=80825,-8752,-24536,-11465,96320,-81994
C00792=80973,-8366,-25985,-11504,97411,-82047
C00793=81511,-5615,-27635,-11617,99868,-82095
C00794=103949,-6271,-30701,-7884,96105,-76175
C00795=129846,-17397,-52274,-16165,101048,-68229
C00796=163642,29140,5761,-44799,70700,-52559
C00797=162591,31494,11671,-45064,68427,-51999
C00798=162048,30394,11874,-43983,65447,-51631
C00799=161982,31813,14334,-41708,59650,-50819
C00800=161467,24519,6374,-40573,59309,-51272
C00801=161788,23282,1722,-39913,61178,-51925
C00802=148843,20256,-8268,-42580,75292,-58905
C00803=147687,21461,-3477,-42608,73008,-58456
C00804=147474,22713,-827,-42735,72168,-58194
C00805=145829,17703,-5538,-42117,71635,-58722
C00806=146103,16605,-8013,-42018,72487,-58958
C00807=147273,15378,-12798,-41999,74773,-59389
C00808=132879,31978,-11069,-11402,105457,-66436
C00809=133021,29093,-9797,-11280,103253,-66180
C00810=131898,46229,9833,-9962,110180,-66921
C00811=130688,40255,3261,-9867,109174,-67217
C00812=130053,42231,5661,-10091,111027,-67639
C00813=131193,25278,-13529,-11136,103347,-66799
C00814=131063,28208,-14820,-11259,105588,-67051
C00815=112468,-32306,-55652,-4896,84919,-46156
C00816=96808,-82585,-76071,-53,68600,-46133
C00817=69953,-63335,-76496,8026,68297,-36882
C00818=96929,-90691,-89138,-5080,61517,23019
C00819=101389,-60822,-75148,-6919,68546,70102
C00820=109578,66950,51259,9202,73878,70224
C00821=119285,73548,61078,7759,54489,67872
C00822=119140,78931,71700,8230,50768,67516
C00823=119625,58082,57992,11126,34581,65932
C00824=123364,68268,69491,7525,32771,67988
C00825=122687,69615,57970,5984,54089,69256
C00826=122770,54503,36545,5592,59480,69583
C00827=119074,82203,59752,14757,75142,72556
C00828=112473,77653,55392,16315,76732,70397
C00829=112597,64720,47818,22234,69078,68724
C00830=113195,66142,49473,22093,68650,68874
C00831=113258,68857,52652,22154,68111,68793
C00832=116388,75351,60395,21391,65952,69596
C00833=116375,72151,56555,21287,66626,69721
C00834=116824,73080,57665,21174,66318,69837
C00835=121396,72779,51526,8459,68942,71502
C00836=127130,57447,36738,757,68697,35525
C00837=129893,63235,47621,-3557,65457,33128
C00838=128808,60089,44122,-3143,65953,32716
C00839=130205,57581,36634,-4742,69462,32000
C00840=130312,54578,33992,-4779,69550,32035
C00841=129992,46081,35923,-20239,67004,-8502
C00842=121835,41418,34711,-6021,59386,-22657
C00843=117745,46484,42710,5309,56994,-25598
C00844=117421,45985,43643,5502,56187,-25765
C00845=128073,50557,47782,-20949,62737,-7811
C00846=128141,51586,49590,-20554,61962,-8032
C00847=121273,40131,39499,-4242,51746,-24031
C00848=122651,35401,27095,-8965,61652,-19959
C00849=109578,66950,51259,9202,73878,70224
C00850=101389,-60822,-75148,-6919,68546,70102
C00851=96929,-90691,-89138,-5080,61517,23019
C00852=93242,-104717,-83164,-3670,50463,-28203
C00853=113023,-47673,-50887,-12494,73990,-34579
C00854=92156,-22649,-39625,-10516,94476,-60392
C00855=92549,-23820,-36378,-10508,91967,-60047
C00856=93168,-23682,-34836,-10551,91183,-59771
C00857=95681,-22921,-34071,-10762,91434,-58934
C00858=94898,-22950,-35761,-10710,92338,-59280
C00859=94492,-21797,-39017,-10723,94837,-59633
C00860=92575,-26977,-42679,-21088,73618,-56030
C00861=92430,-25186,-37423,-21282,71416,-55682
C00862=92878,-24238,-35435,-21526,70842,-55408
C00863=96065,-22906,-34163,-23638,71815,-54341
C00864=95477,-23933,-36320,-23344,72386,-54682
C00865=95719,-25683,-41558,-23174,74597,-55037
C00866=111616,-56743,-62949,-22039,72011,-39056
C00867=96929,-90691,-89138,-5080,61517,-27168
C00868=96929,-90691,-89138,-5080,61517,23019
C00869=101389,-60822,-75148,-6919,68546,70102
C00870=109578,66950,51259,9202,73878,70224
C00871=108278,48890,46404,6655,48460,73563
C00872=108252,54023,56228,7048,45078,73302
C00873=108060,40798,52110,13776,28764,70729
C00874=112800,50045,60477,7453,29903,74191
C00875=112495,52250,52136,4220,46380,75358
C00876=112766,56024,54314,4011,46966,75508
C00877=103660,28975,43016,-10311,30529,75473
C00878=104692,35200,60863,-30413,16065,83251
C00879=105089,39423,66918,-34170,14880,85035
C00880=103103,37348,64656,-29541,14457,82654
C00881=100412,37194,55383,-7603,26828,73795
C00882=100998,29868,43914,-7479,30147,73786
C00883=109578,66950,51259,9202,73878,70224
C00884=101389,-60822,-75148,-6919,68546,70102
C00885=96929,-90691,-89138,-5080,61517,23019
C00886=92414,-106749,-81881,-3283,48598,-28500
C00887=109112,-55837,-56038,-6601,71444,-37060
C00888=90570,-23240,-39845,1682,91658,-61068
C00889=90349,-1837,-19216,4288,101242,-62233
C00890=89876,4658,-11592,5336,104467,-62228
C00891=91883,5295,-10855,6364,104142,-61464
C00892=95291,-22836,-35623,1093,89189,-59526
C00893=94239,-22001,-38963,1226,91687,-59852
C00894=90424,-29050,-43505,-3763,58999,-61302
C00895=86008,-21130,-36360,6353,62529,-61992
C00896=86680,-19135,-33236,6051,61587,-61792
C00897=89871,-18454,-32736,4367,61424,-60601
C00898=95351,-24457,-36663,-6763,57473,-59317
C00899=94707,-27619,-42528,-6252,59394,-59681
C00900=109011,-26713,-50438,-8452,98222,-74634
C00901=131236,23776,-19025,3434,93964,-64709
C00902=130664,38162,-3482,6829,99038,-64158
C00903=130670,46363,8576,7678,101442,-63891
C00904=134671,48665,11259,6610,97243,-62896
C00905=136543,32349,-6519,2125,90508,-63120
C00906=135803,33584,-9338,2313,92894,-63310
C00907=159001,-16036,-30877,-42377,70566,-51510
C00908=152463,-28313,-30724,-35893,55196,-47069
C00909=153151,-16160,-21724,-35569,61642,-49446
C00910=157385,-8578,-13959,-39473,60379,-46999
C00911=158653,-15121,-22520,-39743,62752,-48156
C00912=161766,-5301,-16021,-44095,69224,-49591
C00913=91964,-16840,-43330,-6553,97397,-80206
C00914=99312,-50897,-61026,-22837,72179,-74454
C00915=98138,-49989,-56545,-22703,69739,-74412
C00916=107037,-51945,-50657,-37198,66142,-70452
C00917=99628,-21060,-40506,-23543,91538,-75534
C00918=101911,-27523,-44444,-25592,91744,-74763
C00919=98969,-20169,-40937,-21673,97560,-76394
C00920=97496,-21660,-46096,-18879,96544,-76387
C00921=97638,-23312,-49453,-18962,97729,-76524
C00922=81141,-50558,-66105,-12803,46081,-75388
C00923=80687,-46119,-60183,-12697,44679,-75401
C00924=80513,-44339,-57785,-12667,44105,-75401
C00925=80516,-44488,-54802,-13120,42239,-75121
C00926=80690,-46329,-57233,-13145,42803,-75122
C00927=81145,-50923,-63237,-13239,44177,-75109
C00928=83601,15534,-39616,-9664,96262,-77072
C00929=80484,90945,50155,-4324,118905,-78550
C00930=80490,84570,45509,-4303,118490,-78531
C00931=80493,82108,43801,-4293,118276,-78521
C00932=80495,81630,46278,-4216,116511,-78452
C00933=80492,84058,47940,-4226,116735,-78462
C00934=83493,53381,-2692,-9637,111099,-78940
C00935=91945,-14209,-43630,-9790,83010,-75128
C00936=107113,-96096,-84434,-15453,68738,-68360
C00937=10907,-117335,-90652,18762,63715,59495
C00938=15972,-110889,-128286,10965,59905,43045
BC00000=48813,501269,1075139
BC00001=366895,287876,1075139
BC00002=366895,287876,1075139
BC00003=366895,287876,1075139
BC00004=366895,287876,1075139
BC00005=366895,287876,1075139
BC00006=366895,287876,1075139
BC00007=366895,287876,1075139
BC00008=366895,287876,1075139
BC00009=333040,294697,1075139
BC00010=333040,294697,1075139
BC00011=333040,294697,1075139
BC00012=333040,294697,1075139
BC00013=333040,294697,1075139
BC00014=333040,294697,1075139
BC00015=333040,294697,1075139
BC00016=333040,294697,1075139
BC00017=358075,287887,1075139
BC00018=358075,287887,1075139
BC00019=358075,287887,1075139
BC00020=358075,287887,1075139
BC00021=358075,287887,1075139
BC00022=358075,287887,1075139
BC00023=358075,287887,1075139
BC00024=358075,287887,1075139
BC00025=398158,296006,1075139
BC00026=398158,296006,1075139
BC00027=398158,296006,1075139
BC00028=398158,296006,1075139
BC00029=398158,296006,1075139
BC00030=398158,296006,1075139
BC00031=398158,296006,1075139
BC00032=398158,296006,1075139
BC00033=264887,408839,1075139
BC00034=264887,408839,1075139
BC00035=264888,408840,1075136
BC00036=264888,408840,1075135
BC00037=264888,408840,1075135
BC00038=264888,408840,1075132
BC00039=264888,408840,1075132
BC00040=264888,408840,1075132
BC00041=264888,408840,1075132
BC00042=264888,408840,1075132
BC00043=264888,408840,1075128
BC00044=264887,408839,1075139
BC00045=301248,414295,1075139
BC00046=301248,414295,1075139
BC00047=301248,414295,1075139
BC00048=301248,414295,1075139
BC00049=301248,414295,1075139
BC00050=301248,414295,1075139
BC00051=301248,414295,1075139
BC00052=301248,414295,1075139
BC00053=301248,414295,1075139
BC00054=301248,414295,1075139
BC00055=274219,403900,1075139
BC00056=238656,390224,1075139
BC00057=238656,390224,1075139
BC00058=238656,390224,1075139
BC00059=238656,390224,1075139
BC00060=238656,390224,1075139
BC00061=238656,390224,1075139
BC00062=238656,390224,1075139
BC00063=238656,390224,1075139
BC00064=238656,390225,1075135
BC00065=238656,390225,1075135
BC00066=238656,390224,1075139
BC00067=238656,390224,1075139
BC00068=238656,390224,1075139
BC00069=238656,390224,1075139
BC00070=318247,439655,1075139
BC00071=318247,439655,1075139
BC00072=318247,439655,1075139
BC00073=318247,439655,1075139
BC00074=318247,439655,1075139
BC00075=318247,439655,1075139
BC00076=318247,439655,1075139
BC00077=318247,439655,1075139
BC00078=318247,439655,1075139
BC00079=318247,439655,1075139
BC00080=318247,439655,1075139
BC00081=318247,439655,1075139
BC00082=318247,439655,1075139
BC00083=318247,439655,1075139
BC00084=318247,439655,1075139
BC00085=318247,439655,1075139
BC00086=318247,439655,1075139
BC00087=318247,439655,1075139
BC00088=318247,439655,1075139
BC00089=318247,439655,1075139
BC00090=318247,439655,1075139
BC00091=318247,439655,1075139
BC00092=318247,439655,1075139
BC00093=318247,439655,1075139
BC00094=318247,439655,1075139
BC00095=377098,439655,1075139
BC00096=397798,439655,1075139
BC00097=397798,439655,1075139
BC00098=397798,439655,1075139
BC00099=397798,439655,1075139
BC00100=397798,439655,1075139
BC00101=397798,439655,1075139
BC00102=397798,439655,1075139
BC00103=397798,439655,1075139
BC00104=397798,439655,1075139
BC00105=397798,439655,1075139
BC00106=397798,439655,1075139
BC00107=397798,439655,1075139
BC00108=397798,439655,1075139
BC00109=397798,439655,1075139
BC00110=397798,439655,1075139
BC00111=397798,439655,1075139
BC00112=397798,439655,1075139
BC00113=397798,439655,1075139
BC00114=397798,439655,1075139
BC00115=397798,439655,1075139
BC00116=390344,433324,1075139
BC00117=390344,433324,1075139
BC00118=323680,511522,1075139
BC00119=296258,353406,1075139
BC00120=296258,353406,1075139
BC00121=296258,353406,1075139
BC00122=296258,353406,1075139
BC00123=296258,353406,1075139
BC00124=296258,353406,1075139
BC00125=296258,353406,1075139
BC00126=296258,353406,1075139
BC00127=296258,353406,1075139
BC00128=296258,353406,1075139
BC00129=296258,353406,1075139
BC00130=296258,353406,1075139
BC00131=312199,290121,1075139
BC00132=312199,245824,1075139
BC00133=312199,245824,1075139
BC00134=312199,245824,1075139
BC00135=312199,245824,1075139
BC00136=312199,245824,1075139
BC00137=312199,245824,1075139
BC00138=312199,245824,1075139
BC00139=312199,245824,1075139
BC00140=312199,245824,1075139
BC00141=312199,245824,1075139
BC00142=312199,245824,1075139
BC00143=259283,251148,1075139
BC00144=259283,251148,1075139
BC00145=259283,251148,1075139
BC00146=259283,251148,1075139
BC00147=259283,251148,1075139
BC00148=259283,251148,1075139
BC00149=259283,251148,1075139
BC00150=259283,251148,1075139
BC00151=259283,251148,1075139
BC00152=259283,251148,1075139
BC00153=259283,251148,1075139
BC00154=259283,251148,1075139
BC00155=211515,238198,1075139
BC00156=211515,238198,1075139
BC00157=211515,238198,1075139
BC00158=211515,238198,1075139
BC00159=211515,238198,1075139
BC00160=211515,238198,1075139
BC00161=211515,238198,1075139
BC00162=211515,238198,1075139
BC00163=211515,238198,1075139
BC00164=211515,238198,1075139
BC00165=211515,238198,1075139
BC00166=182487,238237,1075139
BC00167=184353,236726,1075139
BC00168=184353,236710,1075139
BC00169=184317,236583,1075139
BC00170=184881,233559,1075139
BC00171=184317,236583,1075139
BC00172=184735,236445,1075139
BC00173=187871,236988,1075139
BC00174=184735,236445,1075139
BC00175=178206,241731,1075139
BC00176=185188,240150,1075139
BC00177=186084,235310,1075139
BC00178=186442,233366,1075138
BC00179=186443,233357,1075139
BC00180=186562,233334,1075139
BC00181=187125,230310,1075139
BC00182=186562,233334,1075139
BC00183=185308,240110,1075139
BC00184=153065,191986,1075139
BC00185=123072,128894,1075139
BC00186=126316,134328,1075139
BC00187=127614,136496,1075139
BC00188=127614,136486,1075139
BC00189=127614,136502,1075139
BC00190=153737,125360,1075139
BC00191=152136,128016,1075139
BC00192=153737,125360,1075139
BC00193=104350,151955,1075139
BC00194=107104,153499,1075139
BC00195=104350,151955,1075139
BC00196=97474,145929,1075139
BC00197=140327,144391,1075139
BC00198=158627,143734,1075139
BC00199=155448,149073,1075139
BC00200=155090,149654,1075139
BC00201=155090,149646,1075139
BC00202=155272,149742,1075139
BC00203=153671,152398,1075139
BC00204=155272,149742,1075139
BC00205=158875,143812,1075139
BC00206=211321,196495,1075139
BC00207=274607,206177,1075139
BC00208=371745,147058,1075139
BC00209=371745,147058,1075139
BC00210=371745,147058,1075139
BC00211=371745,147058,1075139
BC00212=371745,147058,1075139
BC00213=371745,147058,1075139
BC00214=371745,147058,1075139
BC00215=371745,147058,1075139
BC00216=371745,147058,1075139
BC00217=371745,147058,1075139
BC00218=371745,147058,1075139
BC00219=371745,147058,1075139
BC00220=371745,147058,1075139
BC00221=371745,147058,1075139
BC00222=371745,147058,1075139
BC00223=314169,251254,1075139
BC00224=247655,219498,1075139
BC00225=247655,219498,1075139
BC00226=247655,219498,1075139
BC00227=247655,219498,1075139
BC00228=247655,219498,1075139
BC00229=247655,219498,1075139
BC00230=247655,219498,1075139
BC00231=247655,219498,1075139
BC00232=247655,219498,1075139
BC00233=247655,219498,1075139
BC00234=247655,219498,1075139
BC00235=247655,219498,1075139
BC00236=303021,318054,1075139
BC00237=380976,369454,1075139
BC00238=380976,369454,1075139
BC00239=380976,369454,1075139
BC00240=380976,369454,1075139
BC00241=380976,369454,1075139
BC00242=380976,369454,1075139
BC00243=380976,369454,1075139
BC00244=380976,369454,1075139
BC00245=380976,369454,1075139
BC00246=380976,369454,1075139
BC00247=380976,369454,1075139
BC00248=380976,369454,1075139
BC00249=275240,377785,1075139
BC00250=125700,292206,1075139
BC00251=125700,292206,1075139
BC00252=125700,292206,1075139
BC00253=125700,292206,1075139
BC00254=125700,292206,1075139
BC00255=125700,292206,1075138
BC00256=125700,292206,1075135
BC00257=125700,292206,1075139
BC00258=125700,292206,1075139
BC00259=125700,292206,1075139
BC00260=125700,292206,1075139
BC00261=125700,292206,1075139
BC00262=125700,292206,1075139
BC00263=325003,367566,1075193
BC00264=325003,367566,1075193
BC00265=325003,367566,1075193
BC00266=325003,367566,1075193
BC00267=325003,367566,1075193
BC00268=325003,367566,1075193
BC00269=325003,367566,1075193
BC00270=325003,367566,1075193
BC00271=325003,367566,1075193
BC00272=325003,367566,1075193
BC00273=325003,367566,1075193
BC00274=325003,367566,1075193
BC00275=240651,318179,1075174
BC00276=81319,224890,1075139
BC00277=81319,224890,1075139
BC00278=81319,224890,1075139
BC00279=81319,224890,1075139
BC00280=81319,224890,1075139
BC00281=81319,224890,1075139
BC00282=81319,224890,1075139
BC00283=81319,224890,1075139
BC00284=39875,217643,1075139
BC00285=39875,217643,1075139
BC00286=39875,217643,1075139
BC00287=39875,217643,1075139
BC00288=39875,217643,1075139
BC00289=39875,217643,1075139
BC00290=39875,217643,1075139
BC00291=39875,217643,1075139
BC00292=126048,247985,1075139
BC00293=145702,238926,1075139
BC00294=145702,238926,1075139
BC00295=145702,238926,1075139
BC00296=145702,238926,1075139
BC00297=145702,238926,1075139
BC00298=145702,238926,1075139
BC00299=145702,238926,1075139
BC00300=145702,238926,1075139
BC00301=145702,238926,1075139
BC00302=145702,238926,1075139
BC00303=145702,238926,1075139
BC00304=145702,238926,1075139
BC00305=127177,276102,1075139
BC00306=75481,322634,1075139
BC00307=75481,322634,1075139
BC00308=75481,322634,1075139
BC00309=75481,322634,1075139
BC00310=75481,322634,1075139
BC00311=75481,322634,1075139
BC00312=75481,322634,1075139
BC00313=75481,322634,1075139
BC00314=75481,322634,1075139
BC00315=75481,322634,1075139
BC00316=75481,322634,1075139
BC00317=75481,322634,1075139
BC00318=75481,322634,1075139
BC00319=75481,322634,1075139
BC00320=75481,322634,1075139
BC00321=75481,322634,1075139
BC00322=75481,322634,1075139
BC00323=58814,337696,1075139
BC00324=43258,351755,1075139
BC00325=43258,351755,1075139
BC00326=43258,351755,1075139
BC00327=43258,351755,1075139
BC00328=43258,351755,1075139
BC00329=43258,351755,1075139
BC00330=43258,351755,1075139
BC00331=43258,351755,1075139
BC00332=43258,351755,1075139
BC00333=191423,293819,1075139
BC00334=209577,315616,1075139
BC00335=209577,315616,1075139
BC00336=209577,315616,1075139
BC00337=209577,315616,1075135
BC00338=209577,315616,1075139
BC00339=209577,315616,1075139
BC00340=209200,339183,1075139
BC00341=226850,335636,1075139
BC00342=228819,334245,1075139
BC00343=228819,334245,1075139
BC00344=228818,334247,1075135
BC00345=228818,334246,1075136
BC00346=228819,334245,1075139
BC00347=228819,334245,1075139
BC00348=228819,334245,1075139
BC00349=228819,334245,1075139
BC00350=228819,334245,1075139
BC00351=212667,203752,1075139
BC00352=212667,185592,1075139
BC00353=212231,190237,1075139
BC00354=212130,191331,1075135
BC00355=214778,193391,1075138
BC00356=222170,195981,1075139
BC00357=222606,191336,1075139
BC00358=293461,217046,1075139
BC00359=293461,217046,1075139
BC00360=293461,217046,1075139
BC00361=293461,217046,1075139
BC00362=293461,217046,1075139
BC00363=293461,217046,1075139
BC00364=293461,217046,1075139
BC00365=293461,217046,1075139
BC00366=248761,215697,1075139
BC00367=147608,172175,1075139
BC00368=124934,156734,1075139
BC00369=124934,156734,1075139
BC00370=124934,156734,1075139
BC00371=124934,156734,1075139
BC00372=124934,156734,1075139
BC00373=124934,156734,1075139
BC00374=124934,156734,1075139
BC00375=106662,143944,1075139
BC00376=106662,143944,1075139
BC00377=106662,143944,1075139
BC00378=106662,143944,1075139
BC00379=106662,143944,1075139
BC00380=106662,143944,1075139
BC00381=106662,155705,1075139
BC00382=288347,238792,1075139
BC00383=319864,257821,1075139
BC00384=316187,259932,1075139
BC00385=314717,260776,1075138
BC00386=314716,260777,1075139
BC00387=294125,249227,1075139
BC00388=285335,240623,1075139
BC00389=280828,236212,1075139
BC00390=254340,221178,1075136
BC00391=253980,219316,1075139
BC00392=256761,216362,1075139
BC00393=224898,195450,1075139
BC00394=193391,175353,1075139
BC00395=196536,180842,1075139
BC00396=197049,181737,1075139
BC00397=197381,182312,1075139
BC00398=196536,180831,1075139
BC00399=193391,175343,1075139
BC00400=170860,158975,1075139
BC00401=152991,145993,1075139
BC00402=152991,145993,1075139
BC00403=155583,151896,1075139
BC00404=156620,154258,1075139
BC00405=230582,164381,1075139
BC00406=176880,134401,1075139
BC00407=222677,176979,1075139
BC00408=228168,179508,1075139
BC00409=235185,179594,1075139
BC00410=242581,209775,1075139
BC00411=282664,373339,1075139
BC00412=287377,415944,1075139
BC00413=293850,413917,1075139
BC00414=296439,413107,1075139
BC00415=296321,413021,1075139
BC00416=296321,413021,1075139
BC00417=296321,413021,1075139
BC00418=293584,413723,1075139
BC00419=287111,415750,1075139
BC00420=265157,384983,1075139
BC00421=271825,383261,1075139
BC00422=274492,382572,1075139
BC00423=274492,382572,1075139
BC00424=271826,383216,1075139
BC00425=265158,384938,1075139
BC00426=347759,380452,1075139
BC00427=348420,380650,1075139
BC00428=348684,380729,1075139
BC00429=352817,383042,1075139
BC00430=364797,389762,1075139
BC00431=368926,392082,1075139
BC00432=368661,392003,1075139
BC00433=368000,391805,1075139
BC00434=368000,391805,1075139
BC00435=374651,423539,1075139
BC00436=391328,503109,1075139
BC00437=391328,503109,1075139
BC00438=391328,503109,1075139
BC00439=391328,503109,1075139
BC00440=391328,503109,1075139
BC00441=391328,503109,1075139
BC00442=391328,503109,1075139
BC00443=391328,503109,1075139
BC00444=391328,503108,1075138
BC00445=391328,503109,1075139
BC00446=391328,503109,1075139
BC00447=391328,503109,1075139
BC00448=358857,503109,1075139
BC00449=250155,294085,1075139
BC00450=255354,296197,1075139
BC00451=257433,297042,1075139
BC00452=259835,293058,1075139
BC00453=270486,275398,1075139
BC00454=268406,274554,1075139
BC00455=263207,272441,1075139
BC00456=251679,365603,1075139
BC00457=253900,360561,1075139
BC00458=254788,358544,1075138
BC00459=231432,345511,1075139
BC00460=231432,345511,1075139
BC00461=193281,329322,1075139
BC00462=188554,329982,1075139
BC00463=185285,334773,1075139
BC00464=261316,356567,1075139
BC00465=297096,366823,1075139
BC00466=293507,360766,1075139
BC00467=292071,358344,1075139
BC00468=292072,358325,1075139
BC00469=293507,360744,1075139
BC00470=297096,366801,1075139
BC00471=297096,366823,1075139
BC00472=112329,235363,1075139
BC00473=112329,235363,1075139
BC00474=111530,230597,1075139
BC00475=111210,228691,1075139
BC00476=63682,220459,1075139
BC00477=64002,222365,1075139
BC00478=64801,227131,1075139
BC00479=55513,330800,1075139
BC00480=51579,332061,1075139
BC00481=50005,332565,1075139
BC00482=45879,356917,1075139
BC00483=46055,340308,1075139
BC00484=43971,345622,1075139
BC00485=45459,346376,1075139
BC00486=45459,346376,1075139
BC00487=45459,346376,1075139
BC00488=45459,346376,1075139
BC00489=45459,346376,1075139
BC00490=49366,347783,1075139
BC00491=32175,334569,1075139
BC00492=35183,333207,1075139
BC00493=36386,332662,1075139
BC00494=24154,317654,1075139
BC00495=24100,334244,1075139
BC00496=21697,333868,1075139
BC00497=10090,331721,1075139
BC00498=7091,330415,1075139
BC00499=124149,231378,1075139
BC00500=124461,225905,1075139
BC00501=124586,223716,1075139
BC00502=119883,222901,1075139
BC00503=114643,221993,1075139
BC00504=114518,224182,1075139
BC00505=114206,229656,1075139
BC00506=169481,226749,1075139
BC00507=218439,224175,1075139
BC00508=214415,222148,1075139
BC00509=212806,221337,1075139
BC00510=212806,221337,1075139
BC00511=212806,221337,1075139
BC00512=212806,221337,1075139
BC00513=218328,226790,1075139
BC00514=222352,228818,1075139
BC00515=147308,231841,1075139
BC00516=86334,206095,1075139
BC00517=90701,204719,1075139
BC00518=92225,204354,1075139
BC00519=87933,207931,1075139
BC00520=87933,207931,1075139
BC00521=87933,207931,1075139
BC00522=86186,208482,1075139
BC00523=81819,209859,1075139
BC00524=86334,206095,1075139
BC00525=118170,307260,1075139
BC00526=118297,311064,1075139
BC00527=118347,312586,1075139
BC00528=127335,312613,1075139
BC00529=127284,311091,1075139
BC00530=127157,307287,1075139
BC00531=149515,294377,1075139
BC00532=148233,298842,1075139
BC00533=148018,300627,1075139
BC00534=150070,300618,1075139
BC00535=152272,298825,1075139
BC00536=153553,294359,1075139
BC00537=119286,287990,1075139
BC00538=119424,292460,1075139
BC00539=119479,294248,1075139
BC00540=115958,294219,1075139
BC00541=115903,292431,1075139
BC00542=115765,287961,1075139
BC00543=206834,274416,1075139
BC00544=246621,268498,1075139
BC00545=251225,265487,1075139
BC00546=253066,264282,1075139
BC00547=305610,287542,1075139
BC00548=289507,284753,1075139
BC00549=289507,284753,1075139
BC00550=265981,288415,1075136
BC00551=265766,290089,1075139
BC00552=265230,294276,1075139
BC00553=152789,271435,1075139
BC00554=155628,267409,1075139
BC00555=156764,265799,1075139
BC00556=187125,277004,1075139
BC00557=135483,267954,1075139
BC00558=183860,266265,1075139
BC00559=204587,267200,1075139
BC00560=210051,271155,1075139
BC00561=285477,353851,1075139
BC00562=322658,411530,1075139
BC00563=322658,411530,1075139
BC00564=322658,411530,1075139
BC00565=322658,411530,1075139
BC00566=322658,411530,1075139
BC00567=322658,411530,1075139
BC00568=322658,411530,1075139
BC00569=322658,411530,1075139
BC00570=272539,420945,1075139
BC00571=266463,422086,1075139
BC00572=266463,422086,1075139
BC00573=267463,419870,1071329
BC00574=266783,420774,1075139
BC00575=266463,422086,1075139
BC00576=266463,422086,1075139
BC00577=266463,422086,1075139
BC00578=266463,422086,1075139
BC00579=235968,403705,1075139
BC00580=235968,403705,1075139
BC00581=235968,403705,1075139
BC00582=235968,403705,1075139
BC00583=235968,403705,1075139
BC00584=235968,403705,1075139
BC00585=235968,403705,1075139
BC00586=235968,403705,1075139
BC00587=237187,402741,1075139
BC00588=295006,362715,1075139
BC00589=205685,258924,1075139
BC00590=204796,257891,1075139
BC00591=205655,252480,1075139
BC00592=205999,250316,1075139
BC00593=202530,248347,1075139
BC00594=218277,237314,1075139
BC00595=218450,239623,1075139
BC00596=218882,245393,1075139
BC00597=188210,264707,1075139
BC00598=189282,258005,1075139
BC00599=189712,255325,1075139
BC00600=185359,252882,1075139
BC00601=184930,255563,1075139
BC00602=183858,262264,1075139
BC00603=163240,249581,1075139
BC00604=166744,245232,1075139
BC00605=168145,243492,1075139
BC00606=172944,246185,1075139
BC00607=171543,247924,1075139
BC00608=168039,252273,1075139
BC00609=205588,237933,1075139
BC00610=237359,225800,1075139
BC00611=234842,220095,1075139
BC00612=233835,217813,1075139
BC00613=237392,219487,1075139
BC00614=238410,221660,1075139
BC00615=241123,227449,1075139
BC00616=186179,231259,1075139
BC00617=137514,234633,1075139
BC00618=142324,230418,1075139
BC00619=135201,224052,1075139
BC00620=135201,224052,1075139
BC00621=134384,223577,1075139
BC00622=132247,225161,1075139
BC00623=126952,229147,1075139
BC00624=137514,234633,1075139
BC00625=284854,339782,1075139
BC00626=323088,248514,1075139
BC00627=324420,245120,1075139
BC00628=324953,243763,1075139
BC00629=379843,253270,1075139
BC00630=379310,254627,1075139
BC00631=377978,258021,1075139
BC00632=387009,264306,1075139
BC00633=391855,267678,1075139
BC00634=387117,263921,1075139
BC00635=386182,263175,1075138
BC00636=386182,263175,1075138
BC00637=386182,263175,1075138
BC00638=386182,263175,1075138
BC00639=364780,283240,1075139
BC00640=368854,287926,1075139
BC00641=358141,287701,1075139
BC00642=354860,281457,1075139
BC00643=353548,278959,1075139
BC00644=349122,282807,1075139
BC00645=357556,273175,1075139
BC00646=359162,275355,1075139
BC00647=363177,280805,1075139
BC00648=322742,336521,1075139
BC00649=135423,234905,1075139
BC00650=139936,232261,1075139
BC00651=141741,231203,1075139
BC00652=133024,192287,1075139
BC00653=133049,212626,1075139
BC00654=142080,160489,1075139
BC00655=142682,147059,1075139
BC00656=139311,141641,1075139
BC00657=142682,147059,1075139
BC00658=21198,517278,1075139
BC00659=21198,517278,429866
BC00660=66799,465991,419725
BC00661=110224,417152,337633
BC00662=124980,400556,122247
BC00663=124980,400556,122247
BC00664=124980,400556,122247
BC00665=124980,400556,122247
BC00666=124980,400556,122247
BC00667=124980,400556,122247
BC00668=124980,400556,122247
BC00669=124980,400556,122247
BC00670=124980,400556,122247
BC00671=124980,400556,122247
BC00672=124980,400556,122247
BC00673=124980,400556,122247
BC00674=124980,400556,122247
BC00675=124980,400556,122247
BC00676=124980,400556,122247
BC00677=136713,400556,283945
BC00678=136713,400556,283945
BC00679=136713,400556,283945
BC00680=136713,400556,283945
BC00681=136713,400556,283945
BC00682=136713,400556,283945
BC00683=136713,400556,283945
BC00684=136713,400556,283945
BC00685=136713,400556,283945
BC00686=136713,400556,232066
BC00687=148065,400556,238331
BC00688=154841,400556,249660
BC00689=163178,400556,279134
BC00690=163178,400556,279134
BC00691=163178,400556,279134
BC00692=163178,400556,279134
BC00693=163178,400556,279134
BC00694=163178,400556,279134
BC00695=163178,400556,279134
BC00696=163178,400556,279134
BC00697=163178,400556,279134
BC00698=110224,417152,230098
BC00699=66799,465991,419725
BC00700=66799,519251,419725
BC00701=252749,519251,277295
BC00702=296498,463393,186341
BC00703=322792,429821,131675
BC00704=322792,429821,131675
BC00705=322792,429821,131675
BC00706=322792,429821,131675
BC00707=322792,429821,131675
BC00708=322792,429821,131675
BC00709=322792,429821,131675
BC00710=322792,429821,131675
BC00711=322792,429821,131675
BC00712=303662,400556,204886
BC00713=303662,411227,204886
BC00714=303662,415917,204886
BC00715=303662,415917,204886
BC00716=303662,415917,204886
BC00717=303662,415917,204886
BC00718=303662,400556,204886
BC00719=303662,411314,204886
BC00720=303662,412604,204886
BC00721=343990,442081,139026
BC00722=343990,437458,139026
BC00723=343990,437458,139026
BC00724=343990,437458,139026
BC00725=343990,437458,139026
BC00726=343990,437458,139026
BC00727=343990,437458,139026
BC00728=343990,437458,139026
BC00729=343990,437458,139026
BC00730=300917,439314,218872
BC00731=283877,440048,250459
BC00732=276304,440374,264498
BC00733=276304,440374,264498
BC00734=276304,440374,264498
BC00735=276304,440374,264498
BC00736=276304,440374,264498
BC00737=276304,440374,264498
BC00738=276304,440374,264498
BC00739=276304,440374,264498
BC00740=276304,440374,264498
BC00741=248841,426339,138655
BC00742=248841,426339,138655
BC00743=248841,426339,138655
BC00744=248841,426339,138655
BC00745=248841,426339,138655
BC00746=248841,426339,138655
BC00747=248841,426339,138655
BC00748=248841,426339,138655
BC00749=248841,426339,138655
BC00750=287848,400556,132674
BC00751=287848,400556,132674
BC00752=287848,400556,132674
BC00753=287848,400556,132674
BC00754=287848,400556,132674
BC00755=287848,400556,132674
BC00756=287848,400556,132674
BC00757=287848,400556,132674
BC00758=287848,400556,132674
BC00759=287848,400556,132674
BC00760=287848,400556,132674
BC00761=287848,400556,132674
BC00762=279813,400556,17
BC00763=279813,400556,17
BC00764=279813,400556,17
BC00765=279813,400556,17
BC00766=279813,400556,17
BC00767=279813,400556,17
BC00768=279813,400556,17
BC00769=279813,400556,17
BC00770=279813,400556,17
BC00771=279813,400556,17
BC00772=279813,400556,17
BC00773=279813,400556,17
BC00774=279813,400556,17
BC00775=312308,400556,158769
BC00776=312308,400556,158769
BC00777=312308,400556,158768
BC00778=312308,400556,158769
BC00779=312308,400556,158769
BC00780=312308,400556,158769
BC00781=303066,421715,105063
BC00782=303066,421715,105063
BC00783=303066,421715,105063
BC00784=303066,421715,105063
BC00785=303066,421715,105063
BC00786=303066,421715,105063
BC00787=287852,408667,183289
BC00788=278394,400556,231917
BC00789=278394,400556,231917
BC00790=278394,400556,231917
BC00791=278394,400556,231917
BC00792=278394,400556,231917
BC00793=278394,400556,231917
BC00794=283877,440048,250459
BC00795=300917,439314,218872
BC00796=328923,417583,120701
BC00797=328923,417583,120701
BC00798=328923,417583,120701
BC00799=328923,417583,120701
BC00800=328923,417583,120701
BC00801=328923,417583,120701
BC00802=337213,453034,95368
BC00803=337213,453034,95368
BC00804=337213,453034,95368
BC00805=337213,453034,95368
BC00806=337213,453034,95368
BC00807=337213,453034,95368
BC00808=318162,429946,122343
BC00809=318162,429946,122343
BC00810=318162,429946,122343
BC00811=318162,429946,122343
BC00812=318162,429946,122343
BC00813=318162,429946,122343
BC00814=318162,429946,122343
BC00815=257174,478061,205827
BC00816=245597,487118,221641
BC00817=204965,519251,277295
BC00818=66799,519251,419725
BC00819=66799,465991,419725
BC00820=110224,417152,337633
BC00821=118787,400556,240422
BC00822=118787,400556,240422
BC00823=118787,400556,240422
BC00824=118787,400556,240422
BC00825=118787,400556,240422
BC00826=118787,400556,240422
BC00827=130243,400556,198340
BC00828=110693,400556,198340
BC00829=113235,400556,198340
BC00830=113235,400556,198340
BC00831=113235,400556,198340
BC00832=113235,400556,198340
BC00833=113235,400556,198340
BC00834=113235,400556,198340
BC00835=113235,400556,198340
BC00836=113235,400556,198340
BC00837=113235,400556,198340
BC00838=113235,400556,198340
BC00839=113235,400556,198340
BC00840=113235,400556,228006
BC00841=113235,400556,280256
BC00842=113235,400556,280254
BC00843=113235,400556,280254
BC00844=113235,400556,280254
BC00845=113235,400556,280254
BC00846=113235,400556,280254
BC00847=113235,400556,280254
BC00848=113235,400556,280254
BC00849=110224,417152,337633
BC00850=66799,465991,419725
BC00851=66799,519251,419725
BC00852=252749,519251,277295
BC00853=271419,473397,262334
BC00854=298317,407335,240779
BC00855=298317,407335,240779
BC00856=298317,407335,240779
BC00857=298317,407335,240779
BC00858=298317,407335,240779
BC00859=298317,407335,240779
BC00860=277580,417028,190893
BC00861=277580,417028,190893
BC00862=277580,417028,190893
BC00863=277580,417028,190893
BC00864=277580,417028,190893
BC00865=277580,417028,190893
BC00866=268077,456148,223959
BC00867=252749,519251,277295
BC00868=66799,519251,419725
BC00869=66799,465991,419725
BC00870=110224,417152,337633
BC00871=116529,400556,319233
BC00872=116529,400556,319233
BC00873=116529,400556,319233
BC00874=116529,400556,319233
BC00875=116529,400556,319233
BC00876=116529,400556,319233
BC00877=104242,400556,379272
BC00878=104242,400556,379272
BC00879=104242,400556,379272
BC00880=104242,400556,379272
BC00881=104242,400556,379272
BC00882=104242,400556,379272
BC00883=110224,417152,337633
BC00884=66799,465991,419725
BC00885=66799,539969,419725
BC00886=252749,519251,277295
BC00887=268071,466646,260861
BC00888=286658,402854,240926
BC00889=286659,402854,240926
BC00890=286659,402854,240926
BC00891=286659,402854,240926
BC00892=286658,402854,240926
BC00893=286658,402854,240926
BC00894=267093,432072,158905
BC00895=267093,432072,158905
BC00896=267093,432072,158905
BC00897=267093,432072,158905
BC00898=267093,432072,158905
BC00899=267093,432072,158905
BC00900=283877,440048,250459
BC00901=320500,429384,110898
BC00902=320500,429384,110898
BC00903=320500,429384,110898
BC00904=320500,429384,110898
BC00905=320500,429384,110898
BC00906=320500,429384,110898
BC00907=331313,400556,191260
BC00908=331313,400556,191260
BC00909=331313,400556,191260
BC00910=331313,400556,191260
BC00911=331313,400556,191260
BC00912=331313,400556,191260
BC00913=244057,440048,250459
BC00914=292954,400556,136487
BC00915=292954,400556,136487
BC00916=292954,400556,136487
BC00917=292954,400556,136487
BC00918=292954,400556,136487
BC00919=292954,400557,136484
BC00920=292954,400556,136487
BC00921=292954,400556,136487
BC00922=256479,430691,21535
BC00923=256479,430691,21535
BC00924=256479,430691,21535
BC00925=256479,430691,21535
BC00926=256479,430691,21535
BC00927=256479,430691,21535
BC00928=256059,441499,41693
BC00929=255900,451939,60048
BC00930=255900,451939,60048
BC00931=255900,451939,60048
BC00932=255900,451939,60048
BC00933=255900,451939,60048
BC00934=255900,451939,60048
BC00935=262323,441209,193430
BC00936=262323,441209,193430
BC00937=165804,522273,534000
BC00938=21198,517278,1075139
EC00000=-798156,-1296783
EC00001=-798156,-1296783
EC00002=-798156,-1296783
EC00003=-798156,-1296783
EC00004=-798156,-1296783
EC00005=-798156,-1296783
EC00006=-798156,-1296783
EC00007=-798156,-1296783
EC00008=-798156,-1296783
EC00009=-798156,-1296783
EC00010=-798156,-1296783
EC00011=-798156,-1296783
EC00012=-798156,-1296783
EC00013=-798156,-1296783
EC00014=-798156,-1296783
EC00015=-798156,-1296783
EC00016=-798156,-1296783
EC00017=-798156,-1296783
EC00018=-798156,-1296783
EC00019=-798156,-1296783
EC00020=-798156,-1296783
EC00021=-798156,-1296783
EC00022=-798156,-1296783
EC00023=-798156,-1296783
EC00024=-798156,-1296783
EC00025=-798156,-1296783
EC00026=-798156,-1296783
EC00027=-798156,-1296783
EC00028=-798156,-1296783
EC00029=-798156,-1296783
EC00030=-798156,-1296783
EC00031=-798156,-1296783
EC00032=-798156,-1296783
EC00033=-798156,-1296783
EC00034=-798156,-1296783
EC00035=-798155,-1296782
EC00036=-798155,-1296782
EC00037=-798155,-1296782
EC00038=-798154,-1296781
EC00039=-798154,-1296781
EC00040=-798154,-1296781
EC00041=-798154,-1296781
EC00042=-798154,-1296781
EC00043=-798153,-1296781
EC00044=-798156,-1296783
EC00045=-798156,-1296783
EC00046=-798156,-1296783
EC00047=-798156,-1296783
EC00048=-798156,-1296783
EC00049=-798156,-1296783
EC00050=-798156,-1296783
EC00051=-798156,-1296783
EC00052=-798156,-1296783
EC00053=-798156,-1296783
EC00054=-798156,-1296783
EC00055=-798156,-1296783
EC00056=-798156,-1296783
EC00057=-798156,-1296783
EC00058=-798156,-1296783
EC00059=-798156,-1296783
EC00060=-798156,-1296783
EC00061=-798156,-1296783
EC00062=-798156,-1296783
EC00063=-798156,-1296783
EC00064=-798155,-1296782
EC00065=-798155,-1296782
EC00066=-798156,-1296783
EC00067=-798156,-1296783
EC00068=-798156,-1296783
EC00069=-798156,-1296783
EC00070=-798156,-1296783
EC00071=-798156,-1296783
EC00072=-798156,-1296783
EC00073=-798156,-1296783
EC00074=-798156,-1296783
EC00075=-798156,-1296783
EC00076=-798156,-1296783
EC00077=-798156,-1296783
EC00078=-798156,-1296783
EC00079=-798156,-1296783
EC00080=-798156,-1296783
EC00081=-798156,-1296783
EC00082=-798156,-1296783
EC00083=-798156,-1296783
EC00084=-798156,-1296783
EC00085=-798156,-1296783
EC00086=-798156,-1296783
EC00087=-798156,-1296783
EC00088=-798156,-1296783
EC00089=-798156,-1296783
EC00090=-798156,-1296783
EC00091=-798156,-1296783
EC00092=-798156,-1296783
EC00093=-798156,-1296783
EC00094=-798156,-1296783
EC00095=-798156,-1296783
EC00096=-798156,-1296783
EC00097=-798156,-1296783
EC00098=-798156,-1296783
EC00099=-798156,-1296783
EC00100=-798156,-1296783
EC00101=-798156,-1296783
EC00102=-798156,-1296783
EC00103=-798156,-1296783
EC00104=-798156,-1296783
EC00105=-798156,-1296783
EC00106=-798156,-1296783
EC00107=-798156,-1296783
EC00108=-798156,-1296783
EC00109=-798156,-1296783
EC00110=-798156,-1296783
EC00111=-798156,-1296783
EC00112=-798156,-1296783
EC00113=-798156,-1296783
EC00114=-798156,-1296783
EC00115=-798156,-1296783
EC00116=-798156,-1296783
EC00117=-798156,-1296783
EC00118=-798156,-1296783
EC00119=-798156,-1296783
EC00120=-798156,-1296783
EC00121=-798156,-1296783
EC00122=-798156,-1296783
EC00123=-798156,-1296783
EC00124=-798156,-1296783
EC00125=-798156,-1296783
EC00126=-798156,-1296783
EC00127=-798156,-1296783
EC00128=-798156,-1296783
EC00129=-798156,-1296783
EC00130=-798156,-1296783
EC00131=-798156,-1296783
EC00132=-798156,-1296783
EC00133=-798156,-1296783
EC00134=-798156,-1296783
EC00135=-798156,-1296783
EC00136=-798156,-1296783
EC00137=-798156,-1296783
EC00138=-798156,-1296783
EC00139=-798156,-1296783
EC00140=-798156,-1296783
EC00141=-798156,-1296783
EC00142=-798156,-1296783
EC00143=-798156,-1296783
EC00144=-798156,-1296783
EC00145=-798156,-1296783
EC00146=-798156,-1296783
EC00147=-798156,-1296783
EC00148=-798156,-1296783
EC00149=-798156,-1296783
EC00150=-798156,-1296783
EC00151=-798156,-1296783
EC00152=-798156,-1296783
EC00153=-798156,-1296783
EC00154=-798156,-1296783
EC00155=-798156,-1296783
EC00156=-798156,-1296783
EC00157=-798156,-1296783
EC00158=-798156,-1296783
EC00159=-798156,-1296783
EC00160=-798156,-1296783
EC00161=-798156,-1296783
EC00162=-798156,-1296783
EC00163=-798156,-1296783
EC00164=-798156,-1296783
EC00165=-798156,-1296783
EC00166=-798156,-1296783
EC00167=-798156,-1296783
EC00168=-798156,-1296783
EC00169=-798156,-1296783
EC00170=-798156,-1296783
EC00171=-798156,-1296783
EC00172=-798156,-1296783
EC00173=-798156,-1296783
EC00174=-798156,-1296783
EC00175=-798156,-1296783
EC00176=-798156,-1296783
EC00177=-798156,-1296783
EC00178=-798155,-1296782
EC00179=-798156,-1296783
EC00180=-798156,-1296783
EC00181=-798156,-1296783
EC00182=-798156,-1296783
EC00183=-798156,-1296783
EC00184=-798156,-1296783
EC00185=-798156,-1296783
EC00186=-798156,-1296783
EC00187=-798156,-1296783
EC00188=-798156,-1296783
EC00189=-798156,-1296783
EC00190=-798156,-1296783
EC00191=-798156,-1296783
EC00192=-798156,-1296783
EC00193=-798156,-1296783
EC00194=-798156,-1296783
EC00195=-798156,-1296783
EC00196=-798156,-1296783
EC00197=-798156,-1296783
EC00198=-798156,-1296783
EC00199=-798156,-1296783
EC00200=-798156,-1296783
EC00201=-798156,-1296783
EC00202=-798156,-1296783
EC00203=-798156,-1296783
EC00204=-798156,-1296783
EC00205=-798156,-1296783
EC00206=-798156,-1296783
EC00207=-798156,-1296783
EC00208=-798156,-1296783
EC00209=-798156,-1296783
EC00210=-798156,-1296783
EC00211=-798156,-1296783
EC00212=-798156,-1296783
EC00213=-798156,-1296783
EC00214=-798156,-1296783
EC00215=-798156,-1296783
EC00216=-798156,-1296783
EC00217=-798156,-1296783
EC00218=-798156,-1296783
EC00219=-798156,-1296783
EC00220=-798156,-1296783
EC00221=-798156,-1296783
EC00222=-798156,-1296783
EC00223=-798156,-1296783
EC00224=-798156,-1296783
EC00225=-798156,-1296783
EC00226=-798156,-1296783
EC00227=-798156,-1296783
EC00228=-798156,-1296783
EC00229=-798156,-1296783
EC00230=-798156,-1296783
EC00231=-798156,-1296783
EC00232=-798156,-1296783
EC00233=-798156,-1296783
EC00234=-798156,-1296783
EC00235=-798156,-1296783
EC00236=-798156,-1296783
EC00237=-798156,-1296783
EC00238=-798156,-1296783
EC00239=-798156,-1296783
EC00240=-798156,-1296783
EC00241=-798156,-1296783
EC00242=-798156,-1296783
EC00243=-798156,-1296783
EC00244=-798156,-1296783
EC00245=-798156,-1296783
EC00246=-798156,-1296783
EC00247=-798156,-1296783
EC00248=-798156,-1296783
EC00249=-798156,-1296783
EC00250=-798156,-1296783
EC00251=-798156,-1296783
EC00252=-798156,-1296783
EC00253=-798156,-1296783
EC00254=-798156,-1296783
EC00255=-798156,-1296783
EC00256=-798155,-1296783
EC00257=-798156,-1296783
EC00258=-798156,-1296783
EC00259=-798156,-1296783
EC00260=-798156,-1296783
EC00261=-798156,-1296783
EC00262=-798156,-1296783
EC00263=-798156,-1296783
EC00264=-798156,-1296783
EC00265=-798156,-1296783
EC00266=-798156,-1296783
EC00267=-798156,-1296783
EC00268=-798156,-1296783
EC00269=-798156,-1296783
EC00270=-798156,-1296783
EC00271=-798156,-1296783
EC00272=-798156,-1296783
EC00273=-798156,-1296783
EC00274=-798156,-1296783
EC00275=-798156,-1296783
EC00276=-798156,-1296783
EC00277=-798156,-1296783
EC00278=-798156,-1296783
EC00279=-798156,-1296783
EC00280=-798156,-1296783
EC00281=-798156,-1296783
EC00282=-798156,-1296783
EC00283=-798156,-1296783
EC00284=-798156,-1296783
EC00285=-798156,-1296783
EC00286=-798156,-1296783
EC00287=-798156,-1296783
EC00288=-798156,-1296783
EC00289=-798156,-1296783
EC00290=-798156,-1296783
EC00291=-798156,-1296783
EC00292=-798156,-1296783
EC00293=-798156,-1296783
EC00294=-798156,-1296783
EC00295=-798156,-1296783
EC00296=-798156,-1296783
EC00297=-798156,-1296783
EC00298=-798156,-1296783
EC00299=-798156,-1296783
EC00300=-798156,-1296783
EC00301=-798156,-1296783
EC00302=-798156,-1296783
EC00303=-798156,-1296783
EC00304=-798156,-1296783
EC00305=-798156,-1296783
EC00306=-798156,-1296783
EC00307=-798156,-1296783
EC00308=-798156,-1296783
EC00309=-798156,-1296783
EC00310=-798156,-1296783
EC00311=-798156,-1296783
EC00312=-798156,-1296783
EC00313=-798156,-1296783
EC00314=-798156,-1296783
EC00315=-798156,-1296783
EC00316=-798156,-1296783
EC00317=-798156,-1296783
EC00318=-798156,-1296783
EC00319=-798156,-1296783
EC00320=-798156,-1296783
EC00321=-798156,-1296783
EC00322=-798156,-1296783
EC00323=-798156,-1296783
EC00324=-798156,-1296783
EC00325=-798156,-1296783
EC00326=-798156,-1296783
EC00327=-798156,-1296783
EC00328=-798156,-1296783
EC00329=-798156,-1296783
EC00330=-798156,-1296783
EC00331=-798156,-1296783
EC00332=-798156,-1296783
EC00333=-798156,-1296783
EC00334=-798156,-1296783
EC00335=-798156,-1296783
EC00336=-798156,-1296783
EC00337=-798155,-1296782
EC00338=-798156,-1296783
EC00339=-798156,-1296783
EC00340=-798156,-1296783
EC00341=-798156,-1296783
EC00342=-798156,-1296783
EC00343=-798156,-1296783
EC00344=-798153,-1296781
EC00345=-798154,-1296782
EC00346=-798156,-1296783
EC00347=-798156,-1296783
EC00348=-798156,-1296783
EC00349=-798156,-1296783
EC00350=-798156,-1296783
EC00351=-798156,-1296783
EC00352=-798156,-1296783
EC00353=-798156,-1296783
EC00354=-798155,-1296782
EC00355=-798156,-1296783
EC00356=-798156,-1296783
EC00357=-798156,-1296783
EC00358=-798156,-1296783
EC00359=-798156,-1296783
EC00360=-798156,-1296783
EC00361=-798156,-1296783
EC00362=-798156,-1296783
EC00363=-798156,-1296783
EC00364=-798156,-1296783
EC00365=-798156,-1296783
EC00366=-798156,-1296783
EC00367=-798156,-1296783
EC00368=-798156,-1296783
EC00369=-798156,-1296783
EC00370=-798156,-1296783
EC00371=-798156,-1296783
EC00372=-798156,-1296783
EC00373=-798156,-1296783
EC00374=-798156,-1296783
EC00375=-798156,-1296783
EC00376=-798156,-1296783
EC00377=-798156,-1296783
EC00378=-798156,-1296783
EC00379=-798156,-1296783
EC00380=-798156,-1296783
EC00381=-798156,-1296783
EC00382=-798156,-1296783
EC00383=-798156,-1296783
EC00384=-798156,-1296783
EC00385=-798155,-1296781
EC00386=-798156,-1296783
EC00387=-798156,-1296783
EC00388=-798156,-1296783
EC00389=-798156,-1296783
EC00390=-798155,-1296782
EC00391=-798156,-1296783
EC00392=-798156,-1296783
EC00393=-798156,-1296783
EC00394=-798156,-1296783
EC00395=-798156,-1296783
EC00396=-798156,-1296783
EC00397=-798156,-1296783
EC00398=-798156,-1296783
EC00399=-798156,-1296783
EC00400=-798156,-1296783
EC00401=-798156,-1296783
EC00402=-798156,-1296783
EC00403=-798156,-1296783
EC00404=-798156,-1296783
EC00405=-798156,-1296783
EC00406=-798156,-1296783
EC00407=-798156,-1296783
EC00408=-798156,-1296783
EC00409=-798156,-1296783
EC00410=-798156,-1296783
EC00411=-798156,-1296783
EC00412=-798156,-1296783
EC00413=-798156,-1296783
EC00414=-798156,-1296783
EC00415=-798156,-1296783
EC00416=-798156,-1296783
EC00417=-798156,-1296783
EC00418=-798156,-1296783
EC00419=-798156,-1296783
EC00420=-798156,-1296783
EC00421=-798156,-1296783
EC00422=-798156,-1296783
EC00423=-798156,-1296783
EC00424=-798156,-1296783
EC00425=-798156,-1296783
EC00426=-798156,-1296783
EC00427=-798156,-1296783
EC00428=-798156,-1296783
EC00429=-798156,-1296783
EC00430=-798156,-1296783
EC00431=-798156,-1296783
EC00432=-798156,-1296783
EC00433=-798156,-1296783
EC00434=-798156,-1296783
EC00435=-798156,-1296783
EC00436=-798156,-1296783
EC00437=-798156,-1296783
EC00438=-798156,-1296783
EC00439=-798156,-1296783
EC00440=-798156,-1296783
EC00441=-798156,-1296783
EC00442=-798156,-1296783
EC00443=-798156,-1296783
EC00444=-798155,-1296782
EC00445=-798156,-1296783
EC00446=-798156,-1296783
EC00447=-798156,-1296783
EC00448=-798156,-1296783
EC00449=-798156,-1296783
EC00450=-798156,-1296783
EC00451=-798156,-1296783
EC00452=-798156,-1296783
EC00453=-798156,-1296783
EC00454=-798156,-1296783
EC00455=-798156,-1296783
EC00456=-798156,-1296783
EC00457=-798156,-1296783
EC00458=-798154,-1296783
EC00459=-798156,-1296783
EC00460=-798156,-1296783
EC00461=-798155,-1296782
EC00462=-798156,-1296783
EC00463=-798156,-1296783
EC00464=-798156,-1296783
EC00465=-798156,-1296783
EC00466=-798156,-1296783
EC00467=-798156,-1296783
EC00468=-798156,-1296783
EC00469=-798156,-1296783
EC00470=-798156,-1296783
EC00471=-798156,-1296783
EC00472=-798156,-1296783
EC00473=-798156,-1296783
EC00474=-798156,-1296783
EC00475=-798156,-1296783
EC00476=-798156,-1296783
EC00477=-798156,-1296783
EC00478=-798156,-1296783
EC00479=-798156,-1296783
EC00480=-798156,-1296783
EC00481=-798156,-1296783
EC00482=-798156,-1296783
EC00483=-798156,-1296783
EC00484=-798156,-1296783
EC00485=-798156,-1296783
EC00486=-798156,-1296783
EC00487=-798156,-1296783
EC00488=-798156,-1296783
EC00489=-798156,-1296783
EC00490=-798156,-1296783
EC00491=-798156,-1296783
EC00492=-798156,-1296783
EC00493=-798156,-1296783
EC00494=-798156,-1296783
EC00495=-798156,-1296783
EC00496=-798156,-1296783
EC00497=-798156,-1296783
EC00498=-798156,-1296783
EC00499=-798156,-1296783
EC00500=-798156,-1296783
EC00501=-798156,-1296783
EC00502=-798156,-1296783
EC00503=-798156,-1296783
EC00504=-798156,-1296783
EC00505=-798156,-1296783
EC00506=-798156,-1296783
EC00507=-798156,-1296783
EC00508=-798156,-1296783
EC00509=-798156,-1296783
EC00510=-798156,-1296783
EC00511=-798156,-1296783
EC00512=-798156,-1296783
EC00513=-798156,-1296783
EC00514=-798156,-1296783
EC00515=-798156,-1296783
EC00516=-798156,-1296783
EC00517=-798156,-1296783
EC00518=-798156,-1296783
EC00519=-798156,-1296783
EC00520=-798156,-1296783
EC00521=-798156,-1296783
EC00522=-798156,-1296783
EC00523=-798156,-1296783
EC00524=-798156,-1296783
EC00525=-798156,-1296783
EC00526=-798156,-1296783
EC00527=-798156,-1296783
EC00528=-798156,-1296783
EC00529=-798156,-1296783
EC00530=-798156,-1296783
EC00531=-798156,-1296783
EC00532=-798156,-1296783
EC00533=-798156,-1296783
EC00534=-798156,-1296783
EC00535=-798156,-1296783
EC00536=-798156,-1296783
EC00537=-798156,-1296783
EC00538=-798156,-1296783
EC00539=-798156,-1296783
EC00540=-798156,-1296783
EC00541=-798156,-1296783
EC00542=-798156,-1296783
EC00543=-798156,-1296783
EC00544=-798156,-1296783
EC00545=-798156,-1296783
EC00546=-798156,-1296783
EC00547=-798156,-1296783
EC00548=-798156,-1296783
EC00549=-798156,-1296783
EC00550=-798155,-1296782
EC00551=-798156,-1296783
EC00552=-798156,-1296783
EC00553=-798156,-1296783
EC00554=-798156,-1296783
EC00555=-798156,-1296783
EC00556=-798156,-1296783
EC00557=-798156,-1296783
EC00558=-798156,-1296783
EC00559=-798156,-1296783
EC00560=-798156,-1296783
EC00561=-798156,-1296783
EC00562=-798156,-1296783
EC00563=-798156,-1296783
EC00564=-798156,-1296783
EC00565=-798156,-1296783
EC00566=-798156,-1296783
EC00567=-798156,-1296783
EC00568=-798156,-1296783
EC00569=-798156,-1296783
EC00570=-798156,-1296783
EC00571=-798156,-1296783
EC00572=-798156,-1296783
EC00573=-798156,-1296783
EC00574=-798156,-1296783
EC00575=-798156,-1296783
EC00576=-798156,-1296783
EC00577=-798156,-1296783
EC00578=-798156,-1296783
EC00579=-798156,-1296783
EC00580=-798156,-1296783
EC00581=-798156,-1296783
EC00582=-798156,-1296783
EC00583=-798156,-1296783
EC00584=-798156,-1296783
EC00585=-798156,-1296783
EC00586=-798156,-1296783
EC00587=-798156,-1296783
EC00588=-798156,-1296783
EC00589=-798156,-1296783
EC00590=-798156,-1296783
EC00591=-798156,-1296783
EC00592=-798156,-1296783
EC00593=-798156,-1296783
EC00594=-798156,-1296783
EC00595=-798156,-1296783
EC00596=-798156,-1296783
EC00597=-798156,-1296783
EC00598=-798156,-1296783
EC00599=-798156,-1296783
EC00600=-798156,-1296783
EC00601=-798156,-1296783
EC00602=-798156,-1296783
EC00603=-798156,-1296783
EC00604=-798156,-1296783
EC00605=-798156,-1296783
EC00606=-798156,-1296783
EC00607=-798156,-1296783
EC00608=-798156,-1296783
EC00609=-798156,-1296783
EC00610=-798156,-1296783
EC00611=-798156,-1296783
EC00612=-798156,-1296783
EC00613=-798156,-1296783
EC00614=-798156,-1296783
EC00615=-798156,-1296783
EC00616=-798156,-1296783
EC00617=-798156,-1296783
EC00618=-798156,-1296783
EC00619=-798156,-1296783
EC00620=-798156,-1296783
EC00621=-798156,-1296783
EC00622=-798156,-1296783
EC00623=-798156,-1296783
EC00624=-798156,-1296783
EC00625=-798156,-1296783
EC00626=-798156,-1296783
EC00627=-798156,-1296783
EC00628=-798156,-1296783
EC00629=-798156,-1296783
EC00630=-798156,-1296783
EC00631=-798156,-1296783
EC00632=-798156,-1296783
EC00633=-798156,-1296783
EC00634=-798156,-1296783
EC00635=-798155,-1296783
EC00636=-798155,-1296783
EC00637=-798155,-1296783
EC00638=-798155,-1296783
EC00639=-798156,-1296783
EC00640=-798156,-1296783
EC00641=-798156,-1296783
EC00642=-798156,-1296783
EC00643=-798156,-1296783
EC00644=-798156,-1296783
EC00645=-798156,-1296783
EC00646=-798156,-1296783
EC00647=-798156,-1296783
EC00648=-798156,-1296783
EC00649=-798156,-1296783
EC00650=-798156,-1296783
EC00651=-798156,-1296783
EC00652=-798156,-1296783
EC00653=-798156,-1296783
EC00654=-798156,-1296783
EC00655=-798156,-1296783
EC00656=-798156,-1296783
EC00657=-798156,-1296783
EC00658=-798156,-1296783
EC00659=-798156,-1296783
EC00660=-798156,-1296783
EC00661=-798156,-1296783
EC00662=-798156,-1296783
EC00663=-798156,-1296783
EC00664=-798156,-1296783
EC00665=-798156,-1296783
EC00666=-798156,-1296783
EC00667=-798156,-1296783
EC00668=-798156,-1296783
EC00669=-798156,-1296783
EC00670=-798156,-1296783
EC00671=-798156,-1296783
EC00672=-798156,-1296783
EC00673=-798156,-1296783
EC00674=-798156,-1296783
EC00675=-798156,-1296783
EC00676=-798156,-1296783
EC00677=-798156,-1296783
EC00678=-798156,-1296783
EC00679=-798156,-1296783
EC00680=-798156,-1296783
EC00681=-798156,-1296783
EC00682=-798156,-1296783
EC00683=-798156,-1296783
EC00684=-798156,-1296783
EC00685=-798156,-1296783
EC00686=-798156,-1296783
EC00687=-798156,-1296783
EC00688=-798156,-1296783
EC00689=-798156,-1296783
EC00690=-798156,-1296783
EC00691=-798156,-1296783
EC00692=-798156,-1296783
EC00693=-798156,-1296783
EC00694=-798156,-1296783
EC00695=-798156,-1296783
EC00696=-798156,-1296783
EC00697=-798156,-1296783
EC00698=-798156,-1296783
EC00699=-798156,-1296783
EC00700=-798156,-1296783
EC00701=-798156,-1296783
EC00702=-798156,-1296783
EC00703=-798156,-1296783
EC00704=-798156,-1296783
EC00705=-798156,-1296783
EC00706=-798156,-1296783
EC00707=-798156,-1296783
EC00708=-798156,-1296783
EC00709=-798156,-1296783
EC00710=-798156,-1296783
EC00711=-798156,-1296783
EC00712=-798156,-1296783
EC00713=-798156,-1296783
EC00714=-798156,-1296783
EC00715=-798156,-1296783
EC00716=-798156,-1296783
EC00717=-798156,-1296783
EC00718=-798156,-1296783
EC00719=-798156,-1296783
EC00720=-798156,-1296783
EC00721=-798156,-1296783
EC00722=-798156,-1296783
EC00723=-798156,-1296783
EC00724=-798156,-1296783
EC00725=-798156,-1296783
EC00726=-798156,-1296783
EC00727=-798156,-1296783
EC00728=-798156,-1296783
EC00729=-798156,-1296783
EC00730=-798156,-1296783
EC00731=-798156,-1296783
EC00732=-798156,-1296783
EC00733=-798156,-1296783
EC00734=-798156,-1296783
EC00735=-798156,-1296783
EC00736=-798156,-1296783
EC00737=-798156,-1296783
EC00738=-798156,-1296783
EC00739=-798156,-1296783
EC00740=-798156,-1296783
EC00741=-798156,-1296783
EC00742=-798156,-1296783
EC00743=-798156,-1296783
EC00744=-798156,-1296783
EC00745=-798156,-1296783
EC00746=-798156,-1296783
EC00747=-798156,-1296783
EC00748=-798156,-1296783
EC00749=-798156,-1296783
EC00750=-798156,-1296783
EC00751=-798156,-1296783
EC00752=-798156,-1296783
EC00753=-798156,-1296783
EC00754=-798156,-1296783
EC00755=-798156,-1296783
EC00756=-798156,-1296783
EC00757=-798156,-1296783
EC00758=-798156,-1296783
EC00759=-798156,-1296783
EC00760=-798156,-1296783
EC00761=-798156,-1296783
EC00762=-798156,-1296783
EC00763=-798156,-1296783
EC00764=-798156,-1296783
EC00765=-798156,-1296783
EC00766=-798156,-1296783
EC00767=-798156,-1296783
EC00768=-798156,-1296783
EC00769=-798156,-1296783
EC00770=-798156,-1296783
EC00771=-798156,-1296783
EC00772=-798156,-1296783
EC00773=-798156,-1296783
EC00774=-798156,-1296783
EC00775=-798156,-1296783
EC00776=-798156,-1296783
EC00777=-798156,-1296781
EC00778=-798156,-1296783
EC00779=-798156,-1296783
EC00780=-798156,-1296783
EC00781=-798156,-1296783
EC00782=-798156,-1296783
EC00783=-798156,-1296783
EC00784=-798156,-1296783
EC00785=-798156,-1296783
EC00786=-798156,-1296783
EC00787=-798156,-1296783
EC00788=-798156,-1296783
EC00789=-798156,-1296783
EC00790=-798156,-1296783
EC00791=-798156,-1296783
EC00792=-798156,-1296783
EC00793=-798156,-1296783
EC00794=-798156,-1296783
EC00795=-798156,-1296783
EC00796=-798156,-1296783
EC00797=-798156,-1296783
EC00798=-798156,-1296783
EC00799=-798156,-1296783
EC00800=-798156,-1296783
EC00801=-798156,-1296783
EC00802=-798156,-1296783
EC00803=-798156,-1296783
EC00804=-798156,-1296783
EC00805=-798156,-1296783
EC00806=-798156,-1296783
EC00807=-798156,-1296783
EC00808=-798156,-1296783
EC00809=-798156,-1296783
EC00810=-798156,-1296783
EC00811=-798156,-1296783
EC00812=-798156,-1296783
EC00813=-798156,-1296783
EC00814=-798156,-1296783
EC00815=-798156,-1296783
EC00816=-798156,-1296783
EC00817=-798156,-1296783
EC00818=-798156,-1296783
EC00819=-798156,-1296783
EC00820=-798156,-1296783
EC00821=-798156,-1296783
EC00822=-798156,-1296783
EC00823=-798156,-1296783
EC00824=-798156,-1296783
EC00825=-798156,-1296783
EC00826=-798156,-1296783
EC00827=-798156,-1296783
EC00828=-798156,-1296783
EC00829=-798156,-1296783
EC00830=-798156,-1296783
EC00831=-798156,-1296783
EC00832=-798156,-1296783
EC00833=-798156,-1296783
EC00834=-798156,-1296783
EC00835=-798156,-1296783
EC00836=-798156,-1296783
EC00837=-798156,-1296783
EC00838=-798156,-1296783
EC00839=-798156,-1296783
EC00840=-798156,-1296783
EC00841=-798156,-1296783
EC00842=-798155,-1296782
EC00843=-798155,-1296782
EC00844=-798155,-1296782
EC00845=-798155,-1296782
EC00846=-798155,-1296782
EC00847=-798155,-1296782
EC00848=-798155,-1296782
EC00849=-798156,-1296783
EC00850=-798156,-1296783
EC00851=-798156,-1296783
EC00852=-798156,-1296783
EC00853=-798156,-1296783
EC00854=-798156,-1296783
EC00855=-798156,-1296783
EC00856=-798156,-1296783
EC00857=-798156,-1296783
EC00858=-798156,-1296783
EC00859=-798156,-1296783
EC00860=-798156,-1296783
EC00861=-798156,-1296783
EC00862=-798156,-1296783
EC00863=-798156,-1296783
EC00864=-798156,-1296783
EC00865=-798156,-1296783
EC00866=-798156,-1296783
EC00867=-798156,-1296783
EC00868=-798156,-1296783
EC00869=-798156,-1296783
EC00870=-798156,-1296783
EC00871=-798156,-1296783
EC00872=-798156,-1296783
EC00873=-798156,-1296783
EC00874=-798156,-1296783
EC00875=-798156,-1296783
EC00876=-798156,-1296783
EC00877=-798156,-1296783
EC00878=-798156,-1296783
EC00879=-798156,-1296783
EC00880=-798156,-1296783
EC00881=-798156,-1296783
EC00882=-798156,-1296783
EC00883=-798156,-1296783
EC00884=-798156,-1296783
EC00885=-798156,-1296783
EC00886=-798156,-1296783
EC00887=-798156,-1296783
EC00888=-798156,-1296783
EC00889=-798156,-1296783
EC00890=-798156,-1296783
EC00891=-798156,-1296783
EC00892=-798156,-1296783
EC00893=-798156,-1296783
EC00894=-798156,-1296783
EC00895=-798156,-1296783
EC00896=-798156,-1296783
EC00897=-798156,-1296783
EC00898=-798156,-1296783
EC00899=-798156,-1296783
EC00900=-798156,-1296783
EC00901=-798156,-1296783
EC00902=-798156,-1296783
EC00903=-798156,-1296783
EC00904=-798156,-1296783
EC00905=-798156,-1296783
EC00906=-798156,-1296783
EC00907=-798156,-1296783
EC00908=-798156,-1296783
EC00909=-798156,-1296783
EC00910=-798156,-1296783
EC00911=-798156,-1296783
EC00912=-798156,-1296783
EC00913=-798156,-1296783
EC00914=-798156,-1296783
EC00915=-798156,-1296783
EC00916=-798156,-1296783
EC00917=-798156,-1296783
EC00918=-798156,-1296783
EC00919=-798155,-1296781
EC00920=-798156,-1296783
EC00921=-798156,-1296783
EC00922=-798156,-1296783
EC00923=-798156,-1296783
EC00924=-798156,-1296783
EC00925=-798156,-1296783
EC00926=-798156,-1296783
EC00927=-798156,-1296783
EC00928=-798156,-1296783
EC00929=-798156,-1296783
EC00930=-798156,-1296783
EC00931=-798156,-1296783
EC00932=-798156,-1296783
EC00933=-798156,-1296783
EC00934=-798156,-1296783
EC00935=-798156,-1296783
EC00936=-798156,-1296783
EC00937=-798156,-1296783
EC00938=-798156,-1296783
///POSTYPE BASE
///RECTAN
///RCONF 0,0,0,0,1,0,0,0,0,0,0,0,0,0,0,0,0,0,0,0,0,0,0,0
P00006=2.006,1.622,-0.565,0.0000,0.0000,0.0000
P00021=0.073,2.058,-0.109,0.0000,0.0000,0.0000
P00022=2.006,1.622,-0.565,0.0000,0.0000,0.0000
///RCONF 0,0,0,0,0,0,0,0,0,0,0,0,0,0,0,0,0,0,0,0,0,0,0,0
P00023=-2.957,-4.083,2.762,0.0000,0.0000,0.0000
P00024=-1.466,-0.226,-0.419,0.0000,0.0000,0.0000
P00025=3.643,0.007,-2.585,0.0000,0.0000,0.0000
P00026=2.644,0.055,-2.583,0.0000,0.0000,0.0000
P00027=2.278,0.099,-4.210,0.0000,0.0000,0.0000
P00028=-1.778,-0.182,-2.050,0.0000,0.0000,0.0000
P00029=1.749,4.006,-0.261,0.0000,0.0000,0.0000
P00030=-0.014,-0.768,0.131,0.0000,0.0000,0.0000
P00031=-0.170,0.039,-0.647,0.0000,0.0000,0.0000
P00032=-0.423,0.157,3.222,0.0000,0.0000,0.0000
P00033=0.854,-1.099,3.047,0.0000,0.0000,0.0000
///RCONF 0,0,0,0,1,0,0,0,0,0,0,0,0,0,0,0,0,0,0,0,0,0,0,0
P00034=-8.151,9.743,-4.393,0.0000,0.0000,0.0000
///RCONF 0,0,0,0,0,0,0,0,0,0,0,0,0,0,0,0,0,0,0,0,0,0,0,0
P00035=0.390,-0.027,1.040,0.0000,0.0000,0.0000
P00040=2.716,-0.016,3.014,0.0000,0.0000,0.0000
P00041=-0.109,0.014,0.966,0.0000,0.0000,0.0000
P00042=-0.220,0.371,-0.613,0.0000,0.0000,0.0000
P00043=-0.179,-5.890,-3.227,0.0000,0.0000,0.0000
P00044=-8.560,-7.557,-5.232,0.0000,0.0000,0.0000
P00045=-8.836,-6.632,-1.438,0.0000,0.0000,0.0000
P00046=-7.725,-0.107,-2.878,0.0000,0.0000,0.0000
///RCONF 0,1,0,0,0,0,0,0,0,0,0,0,0,0,0,0,0,0,0,0,0,0,0,0
P00047=0.052,4.745,-6.175,0.0000,0.0000,0.0000
///RCONF 0,0,0,0,0,0,0,0,0,0,0,0,0,0,0,0,0,0,0,0,0,0,0,0
P00048=-10.315,0.035,-3.101,0.0000,0.0000,0.0000
P00049=-9.638,1.690,-2.627,0.0000,0.0000,0.0000
P00050=-0.123,2.174,-1.314,0.0000,0.0000,0.0000
P00051=-5.945,4.696,-10.293,0.0000,0.0000,0.0000
P00052=-0.153,5.586,-7.982,0.0000,0.0000,0.0000
P00053=0.015,-0.644,-4.942,0.0000,0.0000,0.0000
P00054=-0.184,15.039,-0.270,0.0000,0.0000,0.0000
P00061=1211.499,975.999,-261.374,0.5148,35.2356,175.5099
P00062=1205.574,689.500,-262.704,0.5159,35.2461,175.5270
P00063=1197.217,207.358,-268.729,0.4863,35.2395,175.4586
P00071=-2.048,-0.034,-9.092,0.0000,0.0000,0.0000
P00072=-1.595,-0.049,-6.373,0.0000,0.0000,0.0000
P00073=-8.474,-10.331,-11.894,0.0000,0.0000,0.0000
P00074=1.731,-3.007,-10.460,0.0000,0.0000,0.0000
P00088=-8.588,-0.108,-11.097,0.0000,0.0000,0.0000
P00089=5.931,-12.286,-8.772,0.0000,0.0000,0.0000
P00095=-11.943,-14.820,-6.815,0.0000,0.0000,0.0000
P00096=-4.844,-19.262,-10.890,0.0000,0.0000,0.0000
//INST
///DATE 2024/12/02 21:45
///ATTR SC,RW
///GROUP1 RB1,BS1
///GROUP2 ST1
NOP
'X2_8B-21B(90,180)
'
MOVJ C00000 BC00000 VJ=100.00  +MOVJ EC00000 VJ=100.00
'Path S4722
SFTOF3D
MOVJ C00001 BC00001 VJ=100.00  +MOVJ EC00001 VJ=100.00
MOVL C00002 BC00002 V=666.7  +MOVJ EC00002 VJ=100.00
SMOVL C00003 BC00003 V=166.7  +MOVJ EC00003
SREFP 3 C00004 BC00004  +REFP EC00004
CALL JOB:SEARCH-R1-S13D
SET P095 P006
SFTON3D P095
SMOVL C00005 BC00005 V=166.7  +MOVJ EC00005
SREFP 3 C00006 BC00006  +REFP EC00006
CALL JOB:SEARCH-R1-S13D
SET P095 P006
SFTON3D P095
SMOVL C00007 BC00007 V=166.7  +MOVJ EC00007
MOVL C00008 BC00008 V=1000.0  +MOVJ EC00008 VJ=100.00
'EndPath S4722
'Path S4723
SFTOF3D
MOVJ C00009 BC00009 VJ=100.00  +MOVJ EC00009 VJ=100.00
MOVL C00010 BC00010 V=666.7  +MOVJ EC00010 VJ=100.00
SMOVL C00011 BC00011 V=166.7  +MOVJ EC00011
SREFP 3 C00012 BC00012  +REFP EC00012
CALL JOB:SEARCH-R1-S13D
SET P096 P006
SFTON3D P096
SMOVL C00013 BC00013 V=166.7  +MOVJ EC00013
SREFP 3 C00014 BC00014  +REFP EC00014
CALL JOB:SEARCH-R1-S13D
SET P096 P006
SFTON3D P096
SMOVL C00015 BC00015 V=166.7  +MOVJ EC00015
MOVL C00016 BC00016 V=1000.0  +MOVJ EC00016 VJ=100.00
'EndPath S4723
'
'
'Path S4093
SFTOF3D
MOVJ C00017 BC00017 VJ=100.00  +MOVJ EC00017 VJ=100.00
MOVL C00018 BC00018 V=666.7  +MOVJ EC00018 VJ=100.00
SMOVL C00019 BC00019 V=166.7  +MOVJ EC00019
SREFP 3 C00020 BC00020  +REFP EC00020
CALL JOB:SEARCH-R1-S13D
SET P021 P006
SFTON3D P021
SMOVL C00021 BC00021 V=166.7  +MOVJ EC00021
SREFP 3 C00022 BC00022  +REFP EC00022
CALL JOB:SEARCH-R1-S13D
SET P021 P006
SFTON3D P021
SMOVL C00023 BC00023 V=166.7  +MOVJ EC00023
MOVL C00024 BC00024 V=1000.0  +MOVJ EC00024 VJ=100.00
'EndPath S4093
'Path S4094
SFTOF3D
MOVJ C00025 BC00025 VJ=100.00  +MOVJ EC00025 VJ=100.00
MOVL C00026 BC00026 V=666.7  +MOVJ EC00026 VJ=100.00
SMOVL C00027 BC00027 V=166.7  +MOVJ EC00027
SREFP 3 C00028 BC00028  +REFP EC00028
CALL JOB:SEARCH-R1-S13D
SET P022 P006
SFTON3D P022
SMOVL C00029 BC00029 V=166.7  +MOVJ EC00029
SREFP 3 C00030 BC00030  +REFP EC00030
CALL JOB:SEARCH-R1-S13D
